// TwinCAT 3 PLC project basePLC
// ProgramVersion: 3.1.4023.0
// libraries:
//   Tc2_EtherCAT, * (Beckhoff Automation GmbH)
//   Tc2_Standard, * (Beckhoff Automation GmbH)
//   Tc2_SUPS, * (Beckhoff Automation GmbH)
//   Tc2_System, * (Beckhoff Automation GmbH)
//   Tc2_Utilities, * (Beckhoff Automation GmbH)
//   Tc3_MC2_AdvancedHoming, * (Beckhoff Automation GmbH)
//   Tc3_Module, * (Beckhoff Automation GmbH)
//   VisuDialogs, * (System)
//   Tc2_MC2,3.3.27.0,Beckhoff Automation GmbH
// project tree:
//   / GlobalTextList.TcGTLO, PlcTask.TcTTO, Visualization Manager.TcVMO (not stored)
//   GVLs/ GVL_APP.TcGVL
//   POUs/ MAIN.TcPOU
//   tc_mca_std_lib/DUTs/ RestorePosition.TcDUT, ST_AxisConfig.TcDUT, ST_AxisControl.TcDUT, MotionFunctions.TcDUT, ST_AxisInputs.TcDUT, ST_AxisPersistent.TcDUT, ST_GearAxis.TcDUT, ST_AxisStatus.TcDUT, ST_AxisStruct.TcDUT
//   tc_mca_std_lib/GVLs/ GVL.TcGVL
//   tc_mca_std_lib/POUs/ChangeConfig/ FB_ReadFloatParameter.TcPOU, FB_ReadParameterInNc_v1_00.TcPOU, FB_WriteFloatParameter.TcPOU, FB_WriteParameterInNc_v1_00.TcPOU
//   tc_mca_std_lib/POUs/ErrorHandling/ DUT_ErrorState.TcDUT, FB_ErrorSystem.TcPOU, FB_GenericError.TcPOU, FB_NC_Error.TcPOU, FB_TerminalError.TcPOU, ST_ErrorEntry.TcDUT, ST_ErrorSystem.TcDUT
//   tc_mca_std_lib/POUs/Hardware/EtherCAT_Terminals/Analog_Inputs/ EL3174_0002.TcPOU, EL3214.TcPOU, EL3255.TcPOU
//   tc_mca_std_lib/POUs/Hardware/EtherCAT_Terminals/Digital_Inputs/ EL1008.TcPOU, EL1018.TcPOU, EL1252.TcPOU, EL1808.TcPOU, EL1809.TcPOU, EL1819.TcPOU
//   tc_mca_std_lib/POUs/Hardware/EtherCAT_Terminals/Digital_Outputs/ EL2014.TcPOU, EL2252.TcPOU, EL2808.TcPOU, EL2819.TcPOU
//   tc_mca_std_lib/POUs/Hardware/EtherCAT_Terminals/Digital_Outputs/External_Types/ dutEL2521_Ctrl.TcDUT, dutEL2521_Status.TcDUT
//   tc_mca_std_lib/POUs/Hardware/EtherCAT_Terminals/Drives/ EL2522.TcPOU, EL4134.TcPOU, EL7037.TcPOU, EL7041_0052.TcPOU, EL7047.TcPOU, EL7211.TcPOU
//   tc_mca_std_lib/POUs/Hardware/EtherCAT_Terminals/Feedback_Terminals/ EL5002.TcPOU, EL5021.TcPOU, EL5042.TcPOU, EL5101.TcPOU, EL7201.TcPOU
//   tc_mca_std_lib/POUs/Hardware/EtherCAT_Terminals/System/ EK1100.TcPOU, EK1110.TcPOU, EL9410.TcPOU, EL9505.TcPOU
//   tc_mca_std_lib/POUs/Motion/ FB_Axis.TcPOU
//   tc_mca_std_lib/POUs/Motion/Homing/ FB_HomeDirect.TcPOU, FB_HomeFinish.TcPOU, FB_HomePrepare.TcPOU, FB_HomeReadNcVelocities.TcPOU, FB_HomeReadSoftLimEnable.TcPOU, FB_HomeToSwitch.TcPOU, FB_HomeVirtual.TcPOU, FB_HomeWriteNcVelocities.TcPOU, FB_HomeWriteSoftLimEnable.TcPOU, FB_Homing.TcPOU
//   tc_mca_std_lib/POUs/VISUs/ Error_Log_Visu.TcVIS, languageSupport.TcTLO, MainVisu.TcVIS, visuTextLinks.TcTLO
// (motion and I/O tree: see PLC project untitled1)
// real-time tasks:
//   TASK PlcTask: cycle T#10ms, priority 20, ADS port 350
//   TASK PlcTask1: cycle T#10ms, priority 21, ADS port 351
// variable links:

CONFIGURATION basePLC
    RESOURCE PLC ON TwinCAT3
        TASK PlcTask(INTERVAL := T#10ms, PRIORITY := 20);
        PROGRAM MAIN WITH PlcTask : MAIN;
    END_RESOURCE
END_CONFIGURATION

// ---- tc_mca_std_lib/DUTs/RestorePosition.TcDUT
{attribute 'qualified_only'}
{attribute 'strict'}
TYPE RestorePosition :
(
    DontRestore        :=0,
    RestoreWithoutHome :=1
    //RestoreWithHome    :=2
);
END_TYPE

// ---- tc_mca_std_lib/DUTs/ST_AxisConfig.TcDUT
TYPE ST_AxisConfig :
STRUCT

    ///////Axis Parameters//////
    fOverride           :   LREAL := 100;   //Controller override %
    fVelocity           :   LREAL;          //Velocity must be specified, no default used
    fAcceleration       :   LREAL;          //Not all FBs use, need to change this, 0 is NC default
    fDeceleration       :   LREAL;
    fPosition           :   LREAL;          //Used for absolute positioning
    fHomePosition       :   LREAL;          //Used to home to a value other than 0
    nHomeSeq            :   UINT;           //Homing sequence to perform
    eRestorePosition    :   RestorePosition;
    //Restore position of incremental axis after loss of power to the CPU, 0=don't restore, 1=restore but don't home, 2=restore and home

END_STRUCT
END_TYPE

// ---- tc_mca_std_lib/DUTs/ST_AxisControl.TcDUT
TYPE ST_AxisControl :
STRUCT

///////Actions from EPICS/NICOS/////////
    bExecute            :   BOOL;           //Rising edge to execute move absolute
    bReset              :   BOOL;           //Reset axis signal, must be combined with other signals
    bStop               :   BOOL;           //Stop axis movement
    bEnable             :   BOOL;           //Controller enable
    eCommand            :   MotionFunctions;

///////Axis////////
    bJogFwd             :   BOOL;           //Jog forward
    bJogBwd             :   BOOL;           //Jog backward

END_STRUCT
END_TYPE

// ---- tc_mca_std_lib/DUTs/MotionFunctions.TcDUT
{attribute 'qualified_only'}
{attribute 'strict'}
TYPE MotionFunctions :
(
    MoveAbsolute    := 0,
    MoveRelative    :=1,
    Jog             :=2,
    MoveVelocity    :=3,
    MoveModulo      :=4,
    GearIn          :=5,
    GearOut         :=6,
    MultiGearIn     :=7,
    Home            :=10
):=Jog;
END_TYPE

// ---- tc_mca_std_lib/DUTs/ST_AxisInputs.TcDUT
TYPE ST_AxisInputs :
STRUCT

///////Axis Inputs///////
    bLimitFwd   AT %I*  :   BOOL;           //Forward limit switch
    bLimitBwd   AT %I*  :   BOOL;           //Backward limit switch
    bHomeSensor AT %I*  :   BOOL;           //Reference siganl for homing
    bEncLAtch   AT %I*  :   BOOL;           //Reference index signal from inc. enconder

END_STRUCT
END_TYPE

// ---- tc_mca_std_lib/DUTs/ST_AxisPersistent.TcDUT
TYPE ST_AxisPersistent :
STRUCT

    PERSISTENT iPositionAtShutdown : LREAL;
    bMovingAtShutdown   : BOOL;

END_STRUCT
END_TYPE

// ---- tc_mca_std_lib/DUTs/ST_GearAxis.TcDUT
TYPE ST_GearAxis :
STRUCT
    index   :   UINT:=1;    //index of master axis
    ratio   :   LREAL;      //gearing ratio
END_STRUCT
END_TYPE

// ---- tc_mca_std_lib/DUTs/ST_AxisStatus.TcDUT
TYPE ST_AxisStatus :
STRUCT

///////Outputs/Status/////////
    bEnabled            :   BOOL;           //Axis drive enabled
    bWarning            :   BOOL;           //Warning violation (need to be deinfed all the warning stages)
    bBusy               :   BOOL;           //Axis busy
    bDone               :   BOOL;           //Last function block executed successfully
    bHomed              :   BOOL;           //Axis homed
    bFwEnabled          :   BOOL;           //Positive movement of axis is enabled/disabled
    bBwEnabled          :   BOOL;           //Negative movement of axis is enabled/disabled
    fActPosition        :   LREAL;          //Actual position value
    fActVelocity        :   LREAL;          //Actual velocity
    bError              :   BOOL;           //Motion function block has produced error (NC drive not necessarily in error state)
    nErrorID            :   UDINT;          //Motion function block errorID
    bGeared             :   BOOL;           //Axis is an active slave

END_STRUCT
END_TYPE

// ---- tc_mca_std_lib/DUTs/ST_AxisStruct.TcDUT
TYPE ST_AxisStruct :
STRUCT

///////Actions from EPICS/NICOS/////////
///////Axis////////
    control     : ST_AxisControl;

///////Outputs/Status/////////
    status      : ST_AxisStatus;

///////Axis Parameters//////
    config      : ST_AxisConfig;

///////Axis Inputs///////
    inputs      : ST_AxisInputs;

//////Geraing Parameters//////
    //masterAxis        :   UINT:=1;        //Axes[ ] index for master
    //fGearRatioNum     :   LREAL;          //GearIn ratio numerator
    //iGearRatioDen     :   UINT;           //GearIn ratio denominator
///////Axis Ref/////
    Axis                :   AXIS_REF;       //Link NC axis to this

    masterAxis          :   ST_GearAxis;    //Single master axis
    //slaveAxis         :   ARRAY [1..GVL.axisNum]OF ST_GearAxis :=(index:=0, ratio:=0) ;   //Linking single slave axes
    slaveAxisRatio      :   ARRAY [1..GVL_APP.axisNum] OF LREAL;


//////Extra things of original ISIS Structure/////

    //  bSoftLimPosEn       :   BOOL;           //Enable/disable positive direction software limit
    //  bSoftLimNegEn       :   BOOL;           //Enable/disable negative direction software limit
    //bPosLagEn         :   BOOL;           //Enable/disable position lag

    //Gearing parameters

    //masterAxes            :   ARRAY[1..4] OF ST_MasterAxis;   //ST to hold index and ratio for masters    - GearInMultiMaster
    //fDeceleration     :   LREAL;          //Not all FBs use, need to change this, 0 is NC default
    //  Status              : ST_AxisStatus;
END_STRUCT
END_TYPE

// ---- tc_mca_std_lib/POUs/ErrorHandling/DUT_ErrorState.TcDUT
{attribute 'qualified_only'}
{attribute 'strict'}
TYPE DUT_ErrorState :
(
    None,
    Active,
    Inactive,
    Acknowledged
);
END_TYPE

// ---- tc_mca_std_lib/POUs/ErrorHandling/ST_ErrorEntry.TcDUT
TYPE ST_ErrorEntry :
STRUCT
    ErrorNum    : ULINT := 0;               //ID of the Error entry
    ErrorState  : DUT_ErrorState;           //State of the error

    //Error related
    iTerminalID     : INT;                  //ID of the terminal
    sDateTimeOn     : STRING(24);           //Date and time when the error occured
    sDateTimeOff    : STRING(24);           //Date and time when the error disapeared
    sErrorMessage   : STRING (128);         //Description of the event

    ErrorPriority   : INT;                  //Priority of the error
END_STRUCT
END_TYPE

// ---- tc_mca_std_lib/POUs/ErrorHandling/ST_ErrorSystem.TcDUT
TYPE ST_ErrorSystem :
STRUCT
    //Array of error data. Size = cSizeOfErrorData in the GVL
    aErrorData      : ARRAY [0..cSizeOfErrorData - 1] OF ST_ErrorEntry;     //Error Entry List
    nNextErrorNum   : ULINT := 1;                   //ErrorID for the next error entry
    nNoError        : UINT;                         //Number of errors in the list
    nNoActive       : UINT;                         //Number of Active errors
    nNoInactive     : UINT;                         //Number on Inactive errors
    nNoFree         : UINT;                         //Number of free entries in the list
    nNoOverflow     : INT := 0;                     //Number of overflows. How many error entries have been lost due to the size of the array
END_STRUCT
END_TYPE

// ---- tc_mca_std_lib/POUs/Hardware/EtherCAT_Terminals/Digital_Outputs/External_Types/dutEL2521_Ctrl.TcDUT
TYPE dutEL2521_Ctrl :
STRUCT
    ///The control word (CW) is located in the output process image, and is transmitted from the controller to the terminal.
    ///CW.0 FREQ_SEL 0bin / 1bin  Rapid change of the base frequency (only if the ramp function is inactive):
    ///0bin = Base frequency 1 (object 8001:02)
    ///1bin = Base frequency 2 (object 8001:03)
    FREQ_SEL: BOOL;
    ///CW.1 RAMP_DIS 1bin Operation of the ramp function is cancelled, in spite of object 8000:06 being active; if travel distance control is active, it is interrupted by this bit
    RAMP_DIS: BOOL;
    ///CW.2 GO_COUNTER 1bin  If travel distance control is active (object 8000:0A), then a pre-set counter value is approached when the bit is set
    GO_COUNTER: BOOL;
    ///CW.5 CNT_CLR 1bin The contents of the counter is cleared or set (object 8000:0B) by this bit.
    ///Any overflow or underflow bits that might be set are also cleared by this bit.
    ///The process can be edge triggered or level triggered (object 8000:05).
    CNT_CLR: BOOL;
END_STRUCT
END_TYPE

// ---- tc_mca_std_lib/POUs/Hardware/EtherCAT_Terminals/Digital_Outputs/External_Types/dutEL2521_Status.TcDUT
TYPE dutEL2521_Status :
STRUCT
    ///The status word (SW) is located in the input process image, and is transmitted from the terminal to the controller.
    ///SW.0 SEL_ACK/END_COUNTER 1bin  Confirms the change of base frequency. At activated travel distance control: target counter value reached
    SEL_ACK: BOOL;
    ///SW.1 RAMP_ACTIVE 1bin Ramp is currently being followed
    RAMP_ACTIVE: BOOL;
    ///SW.2 UNDERFLOW 1bin This bit is set if the 16-bit counter underflows (0 -> 65535). It is reset when the counter drops below two thirds of its measuring range (43690 -> 43689) or immediately an overflow occurs.
    UNDERFLOW: BOOL;
    ///SW.3 OVERFLOW 1bin This bit is set if the 16-bit counter overflows (65535 -> 0). It is reset when the counter exceeds one third of its measuring range (21845 -> 21846) or immediately an underflow occurs
    OVERFLOW: BOOL;
    ///SW.4 INPUT_T 1bin Status of INPUT_T
    INPUT_T: BOOL;
    ///SW.5 INPUT_Z 1bin Status of INPUT_Z
    INPUT_Z: BOOL;
    ///SW.6 ERROR 1bin General error bit, included with overflow/underflow
    ERROR: BOOL;
END_STRUCT
END_TYPE

// ---- GVLs/GVL_APP.TcGVL
{attribute 'qualified_only'}
VAR_GLOBAL

END_VAR

VAR_GLOBAL CONSTANT
    axisNum :   UINT:=2;
    //axisCoupleMax :   UINT:=4;
END_VAR

// ---- tc_mca_std_lib/GVLs/GVL.TcGVL
VAR_GLOBAL
    stErrorSystemCom    : ST_ErrorSystem;
    axes            :   ARRAY [1..GVL_APP.axisNum] OF ST_AxisStruct;    //Global array of axisControl structure for holding axis parameters and controls
    iAxis           :   UINT;                                           //Index for running axis

END_VAR

VAR_GLOBAL CONSTANT
    cSizeOfErrorData : UINT := 256;
END_VAR

VAR_GLOBAL PERSISTENT
    axesPersistent  : ARRAY [1..gvl_app.axisNum] OF ST_AxisPersistent;
END_VAR

// ---- POUs/MAIN.TcPOU
PROGRAM MAIN
VAR
    sVersion: STRING:='1.0.0';
    i : UINT; //index variable for AXES()
    aFbAxes: ARRAY [1..gvl_app.axisNum] OF FB_Axis;
    hmiAxisSelection    :   INT:=1;     //Not possible to use local hmi variables for array indexes

(******Outputs: Power for Limit switches and Home Sensors (every 4th output)********)

    bOutput1 AT %Q*: BOOL:= TRUE;
    //bOutput2 AT %Q*: BOOL:= TRUE;
    //bOutput3 AT %Q*: BOOL:= TRUE;
    //bOutput4 AT %Q*: BOOL:= TRUE;
    //bOutput5 AT %Q*: BOOL:= TRUE;
    //bOutput6 AT %Q*: BOOL:= TRUE;
    //bOutput7 AT %Q*: BOOL:= TRUE;
    //bOutput8 AT %Q*: BOOL:= TRUE;
    //bOutput9 AT %Q*: BOOL:= TRUE;
    //bOutput13 AT %Q*: BOOL:= TRUE;
    //bOutput17 AT %Q*: BOOL:= TRUE;
    //bOutput21 AT %Q*: BOOL:= TRUE;
    //bOutput24 AT %Q*: BOOL:= TRUE;
    //bOutput28 AT %Q*: BOOL:= TRUE;

(******Error Handling********)
    fbErrorSystem: FB_ErrorSystem;
    aFbAxesError: ARRAY [1..gvl_app.axisNum] OF FB_NC_Error;

    //fbEL1018  : EL1018;
    //fbEL2808  : EL2808;
    //fbEL5101  : EL5101;
    //fbEL9505  : EL9505;
    //fbEL1252  : EL1252;
    //fbEL9410  : EL9410;
    //fbEL7037  : EL7037;
    //fbEK1110  : EK1110;

(******Startup, Shutdown and UPS********)
    fbUPS                  : FB_S_UPS_CX51x0;
    eUpsMode               : E_S_UPS_Mode   := eSUPS_WrPersistData_Shutdown;
    eStartUp: (ColdStart, ReadAxisFeedbackType, CheckReadDone, ExecuteRestore, CheckRestore, FinishRestore);
    bPositionRestoreDone   : BOOL := FALSE;
    bRestoreExecute        : BOOL := FALSE;
    bExecuteReadEncRefSys  : BOOL := FALSE;
    iRetry                 : INT;
    fbReadEncRefSys        : ARRAY [1..gvl_app.axisNum] OF MC_ReadParameter;
    fbRestorePosition      : ARRAY [1..GVL_app.axisNum] OF MC_SetPosition;

END_VAR

VAR PERSISTENT
    bRestoreOnStartup : BOOL;
END_VAR

fbUPS(eUpsMode := eUpsMode); (* call UPS-FB instance in first lines of the fastest PLC Task *)

IF eGlobalSUpsState = eSUPS_PowerFailure THEN
    (* first cycle of powerfailure *)
    (* execute code that should only be done once with each powerfailure, i.e. increase powerfailure counter *)
    bRestoreOnStartup:=TRUE;
    STORE_PERSISTENT();
    RETURN;
ELSIF eGlobalSUpsState > eSUPS_PowerFailure THEN
    (* next cycles of powerfailure *)
    (* skip regular code execution for the remaining cycles of the powerfailure/writing of persistent data/quick shutdown  ... *)
    RETURN;
END_IF

RESTORE_POSITIONS();
PROG();
AXES();
ERROR();

ACTION AXES:
FOR GVL.iAxis:=1 TO gvl_app.axisNum DO
    aFbAxes[GVL.iAxis](stAxisStruct:=gvl.axes[GVL.iAxis]);
END_FOR
END_ACTION

ACTION ERROR:
//
(****FB containting the log of the errors****)
//
fbErrorSystem(
    En:= TRUE,
    bReset:= ,
    nErrorNum:= ,
    bACK:= ,
    bValidSelection:= ,
    nTableRowIndex:= ,
    EnO=> ,
    nSelectedError=> ,
    pErrorSystem=> );


FOR GVL.iAxis:=1 TO gvl_app.axisNum DO
    aFbAxesError[gvl.iAxis](EN:=TRUE,
    nNC_ErrorID:= gvl.axes[gvl.iAxis].status.nErrorID,
    nNC_AxisID:=gvl.axes[gvl.iAxis].Axis.NcToPlc.AxisId,
    ErrorSystem:= fbErrorSystem.pErrorSystem);
END_FOR



(*call all the necessary instance (input assistance F2 or right click) according to the terminals that you have in your hardware and
 add "TRUE" in the input En, the corresponding number of termianl to the iTerminal_ID and
the variable "fbErrorSystem.pErrorSystem" to the input ErrorSystem in each FB E. g. :
fbEL1808(
    En:= TRUE,
    iTerminal_ID:= 01,
    ErrorSystem:= fbErorSystem.pErrorSystem,
    EnO=> ,
    bError=> );
 *)
END_ACTION

ACTION PROG:
//
(* Program any sequence, safety or feature (if necessary) application specific in thsi section*)

//
END_ACTION

ACTION RESTORE_POSITIONS:
///#########################################################
// This ACT will restore the position of an incremental axis on startup with the act position it read before losing power.
// It checks the type of axis, 0=incremental, and that the axis was stationary at shut down.
// Because 0 equates to incremental we also need to check that the data is valid, otherwise by default it would restore all axes.
// By default an axis will not restore the position unless it is set to opt-in, i.e. gvl.axes[i].config.eRestorePosition is non-zero.
// This needs to be initialised somewhere in TwinCAT code otherwise it will not be available at start up.
// A restore will only be performed on a loss of power, this code shouldn't make any changes on a reset cold, a rest origin or a download.
// There is a enum to allow for different types of restore modes, currently only one is implemented.
// 0 'DontRestore'
// 1 'RestoreWithoutHome' -restores the position using a set position fb and does not set the home bit in the axis struct.
// Note from Beckhoff: "A maximum of 1 MB persistent data can be reliably saved over the entire service life."
///#########################################################

IF bRestoreOnStartup THEN
    bRestoreOnStartup:=FALSE;
    bRestoreExecute:=TRUE;
END_IF

// Upon startup bPositionRestoreDone will be set to FALSE, after successfully completing the following code it will be set TRUE
// and should stay TRUE for the rest of the time the PLC is operational, thus this routine should only be completed once.
IF bRestoreExecute AND NOT bPositionRestoreDone THEN

    // Cycle through function blocks that read the encoder reference system i.e. whether axis is incremental or absolute
    // Result stored in Value, 0=Inc 1=Abs, execute set during the case statement
    FOR i:=1 TO gvl_app.axisNum DO
        fbReadEncRefSys[i](
          Axis:= gvl.axes[i].Axis,
          Enable:= bExecuteReadEncRefSys,
          ParameterNumber:= MC_AxisParameter.AxisEncoderReferenceSystem,
          Value=>,
          ReadMode:= E_READMODE.READMODE_ONCE);
    END_FOR

    // Cycle through set position function blocks for each axis
    FOR i:=1 TO gvl_app.axisNum DO
        fbRestorePosition[i](
         Axis:= gvl.axes[i].Axis,
         Execute:= ,
         Position:= axesPersistent[i].iPositionAtShutdown);
    END_FOR

    CASE eStartUp OF
        ColdStart:
        // First cycle of the PLC, do nothing just give one cycle for variables to initialise
            IF NOT bPositionRestoreDone THEN
                eStartUp:=eStartUp+1;
                iRetry:=0;
            END_IF

        ReadAxisFeedbackType:
        // Exectute the function blocks to read the encoder reference system (0=inc OR 1=ABS)
            bExecuteReadEncRefSys:=TRUE;
            eStartUp:=eStartUp+1;

        CheckReadDone:
        // Check the encoder reference system has been read for all axis -> if busy then continue with PLC cycle and check again next time.
        // If fbReadEncRefSys not started then go back a step.
        // If any axes result in an error the code will get stuck here, this happens if gvl_app.axisNum is not set correctly
            FOR i:=1 TO gvl_app.axisNum DO
                IF fbReadEncRefSys[i].Valid = FALSE THEN
                    IF fbReadEncRefSys[i].Busy = TRUE THEN
                        // Exit MAIN.STARTUP Action and wait till next cycle, needs to cycle through whole program in order for data to update
                        RETURN;
                    ELSE
                        // Sometimes the code gets here and the fbReadEncRefSys[i] misses the rising edge. If  the code gets here it means
                        // .valid=FALSE and .busy=FALSE which indicateds the FB probably hasn't started and thus needs to see a rising edge.
                        // Set execute to low, Exit MAIN.STARTUP and go back a step in the CASE statement.
                        bExecuteReadEncRefSys:=FALSE;
                        eStartUp:=eStartUp-1;
                        iRetry:=iRetry+1; // counter used for troubleshooting to see how many cycles it takes before fbReadEncRefSys function blocks are read correctly
                        RETURN;
                    END_IF
                END_IF
            END_FOR
            // If the code gets here all axes either have .valid=TRUE for all axes
            eStartUp:=eStartUp+1;

        ExecuteRestore:
        // Execute position restore by setting fbRestorePosition.execute = TRUE
            FOR i:=1 TO gvl_app.axisNum DO
                IF fbReadEncRefSys[i].Valid = TRUE AND fbReadEncRefSys[i].Value = 0 AND NOT(axesPersistent[i].bMovingAtShutdown) THEN
                    IF GVL.axes[i].config.eRestorePosition = RestorePosition.RestoreWithoutHome THEN
                        fbRestorePosition[i].Execute:=TRUE;
                    END_IF
                END_IF
            END_FOR
            eStartUp:=eStartUp+1;

        CheckRestore:
        // Check the set position fbs are finished
        // Nothing actually happens if the restore is not done, the code just returns from here each cycle and the
        // bPositionRestoreDone will never get set to TRUE and will take up cycle time
            FOR i:=1 TO gvl_app.axisNum DO
                IF fbReadEncRefSys[i].Valid = TRUE AND fbReadEncRefSys[i].Value = 0 AND NOT(axesPersistent[i].bMovingAtShutdown) THEN
                    IF GVL.axes[i].config.eRestorePosition = RestorePosition.RestoreWithoutHome THEN
                        IF NOT fbRestorePosition[i].Done THEN
                            RETURN;
                        END_IF
                    END_IF
                END_IF
            END_FOR
            eStartUp:=eStartUp+1;

        FinishRestore:
        // Remove execute = TRUE for fbRestorePosition
            FOR i:=1 TO gvl_app.axisNum DO
                fbRestorePosition[i].Execute:=FALSE;
            END_FOR
            bPositionRestoreDone:=TRUE;
            bRestoreExecute:=FALSE;
    END_CASE
END_IF
END_ACTION

ACTION STORE_PERSISTENT:
FOR i:=1 TO gvl_app.axisNum DO
    axesPersistent[i].iPositionAtShutdown:=gvl.axes[i].Axis.NcToPlc.ActPos;
    IF gvl.axes[i].Axis.NcToPlc.ActVelo <> 0 THEN
        axesPersistent[i].bMovingAtShutdown:=TRUE;
    ELSE
        axesPersistent[i].bMovingAtShutdown:=FALSE;
    END_IF
    axesPersistent[i].bMovingAtShutdown:=axesPersistent[i].bMovingAtShutdown OR gvl.axes[i].Axis.Status.Moving;
END_FOR
END_ACTION

END_PROGRAM

// ---- tc_mca_std_lib/POUs/Motion/FB_Axis.TcPOU
///#########################################################
///Function block to run a virtual drive with Nc
/// Library:
/// Tc2_MC2.lib
///
/// Global Variables:
///
/// Data types:
///
/// External functions:
///
///###########################################################
FUNCTION_BLOCK FB_Axis
VAR
    sVersion: STRING:='1.0.4';
    masterAxis          :   ST_GearAxis :=(index:=1, ratio:=0) ;

    i: UINT;
END_VAR
VAR_INPUT

END_VAR
VAR_OUTPUT

END_VAR

VAR_IN_OUT
    stAxisStruct: ST_AxisStruct;
END_VAR
VAR
    fbReset: MC_Reset;
    fbPower: MC_Power;
    fbStop: MC_Stop;
    fbHalt: MC_Halt;
    fbJog: MC_Jog;
    fbMoveAbsolute: MC_MoveAbsolute;
    fbMoveVelocity: MC_MoveVelocity;
    fbMoveRelative: MC_MoveRelative;
    fbMoveModulo: MC_MoveModulo;
    fbGearIn: MC_GearIn;
    fbGearOut: MC_GearOut;
    fbHome: FB_Homing;
    fbExecuteRiseEdge: R_TRIG;
    fbStopRiseEdge: R_TRIG;
    fbResetRiseEdge: R_TRIG;
END_VAR

stAxisStruct.Axis.ReadStatus();

////Call of all MC Instances//////

fbPower(Axis:=stAxisStruct.Axis);
fbPower.Enable:= FALSE;
fbReset(Axis:=stAxisStruct.Axis);
fbReset.Execute:= FALSE;
fbStop(Axis:=stAxisStruct.Axis);
fbStop.Execute:=FALSE;
fbHalt(Axis:=stAxisStruct.Axis);
fbHalt.Execute:=FALSE;
fbJog(Axis:=stAxisStruct.Axis);
fbHome(Axis:=stAxisStruct.Axis);
fbHome.bExecute:=FALSE;
fbMoveAbsolute(Axis:=stAxisStruct.Axis);
fbMoveAbsolute.Execute:=FALSE;
fbMoveRelative(Axis:=stAxisStruct.Axis);
fbMoveRelative.Execute:=FALSE;
fbMoveVelocity(Axis:=stAxisStruct.Axis);
fbMoveVelocity.Execute:=FALSE;
fbMoveModulo(Axis:=stAxisStruct.Axis);
fbMoveModulo.Execute:=FALSE;
fbGearin(Slave:= stAxisStruct.Axis, Master:= GVL.axes[masterAxis.index].Axis);
fbGearIn.Execute:=FALSE;
fbGearOut(Slave:=stAxisStruct.Axis);
fbGearOut.Execute:=FALSE;

stAxisStruct.status.bFwEnabled:= stAxisStruct.inputs.bLimitFwd;
stAxisStruct.status.bBwEnabled:= stAxisStruct.inputs.bLimitBwd;

FOR i:= 1 TO GVL_APP.axisNum DO
    IF (stAxisStruct.slaveAxisRatio[i]<>0) THEN
        stAxisStruct.status.bFwEnabled:=stAxisStruct.status.bFwEnabled AND SEL(stAxisStruct.slaveAxisRatio[i]>0, GVL.axes[i].status.bBwEnabled, GVL.axes[i].status.bFwEnabled);
        stAxisStruct.status.bBwEnabled:=stAxisStruct.status.bBwEnabled AND SEL(stAxisStruct.slaveAxisRatio[i]>0, GVL.axes[i].status.bFwEnabled, GVL.axes[i].status.bBwEnabled);
    END_IF
END_FOR

(*Power*)
    fbPower.Enable:=stAxisStruct.control.bEnable;
    fbPower.Enable_Positive:= stAxisStruct.status.bFwEnabled;
    fbPower.Enable_Negative:= stAxisStruct.status.bBwEnabled;
    fbPower.Override:= stAxisStruct.config.fOverride;
    stAxisStruct.status.bEnabled:=fbPower.Status;

(*Stop*)
    fbStop.Execute:= stAxisStruct.control.bStop;
    fbStop.Deceleration:= stAxisStruct.config.fDeceleration;

IF stAxisStruct.control.bStop AND stAxisStruct.Axis.Status.Stopping THEN
    stAxisStruct.control.bStop:=FALSE;
END_IF

(*Reset*)
    fbReset.Execute:=stAxisStruct.control.bReset AND stAxisStruct.status.bError;

IF stAxisStruct.control.bReset AND NOT (stAxisStruct.status.bError OR stAxisStruct.status.bWarning) THEN
    stAxisStruct.control.bReset:=FALSE;
END_IF

CASE stAxisStruct.control.eCommand OF
    MotionFunctions.MoveAbsolute:
        fbMoveAbsolute.Execute:=stAxisStruct.control.bExecute;
        fbMoveAbsolute.Position:=stAxisStruct.config.fPosition;
        fbMoveAbsolute.Velocity:=ABS(stAxisStruct.config.fVelocity);
        fbMoveAbsolute.Acceleration:=stAxisStruct.config.fAcceleration;
        fbMoveAbsolute.Deceleration:=stAxisStruct.config.fDeceleration;

    MotionFunctions.MoveRelative:
        fbMoveRelative.Execute:=stAxisStruct.control.bExecute;
        fbMoveRelative.Distance:=stAxisStruct.config.fPosition;
        fbMoveRelative.Velocity:=ABS(stAxisStruct.config.fVelocity);
        fbMoveRelative.Acceleration:=stAxisStruct.config.fAcceleration;
        fbMoveRelative.Deceleration:=stAxisStruct.config.fDeceleration;

    MotionFunctions.Jog:
        fbJog.JogForward:=stAxisStruct.control.bJogFwd AND NOT (stAxisStruct.control.bExecute OR stAxisStruct.status.bError);
        fbJog.JogBackwards:=stAxisStruct.control.bJogBwd AND NOT (stAxisStruct.control.bExecute OR stAxisStruct.status.bError);
        fbJog.Mode:=0;
        fbJog.Velocity:=stAxisStruct.config.fVelocity;
        fbJog.Acceleration:=stAxisStruct.config.fAcceleration;
        fbJog.Deceleration:=stAxisStruct.config.fDeceleration;

    MotionFunctions.MoveVelocity:
        fbMoveVelocity.Execute:=stAxisStruct.control.bExecute;
        fbMoveVelocity.Velocity:=ABS(stAxisStruct.config.fVelocity);
        fbMoveVelocity.Acceleration:=stAxisStruct.config.fAcceleration;
        fbMoveVelocity.Deceleration:=stAxisStruct.config.fDeceleration;
        fbMoveVelocity.Direction:=SEL(stAxisStruct.config.fVelocity<0, MC_Positive_Direction, MC_Negative_Direction);

    MotionFunctions.Movemodulo:
        fbMoveModulo.Execute:=stAxisStruct.control.bExecute;
        fbMoveModulo.Position:=stAxisStruct.config.fPosition;
        fbMoveModulo.Velocity:=ABS(stAxisStruct.config.fVelocity);
        fbMoveModulo.Acceleration:=stAxisStruct.config.fAcceleration;
        fbMoveModulo.Deceleration:=stAxisStruct.config.fDeceleration;


    MotionFunctions.GearIn:
        fbGearIn.Execute:=          stAxisStruct.control.bExecute;
        fbGearIn.RatioNumerator:=   masterAxis.Ratio;
        fbGearIn.RatioDenominator:=1;       //kept static as numerator is LREAL and consistent with multigearing

        IF NOT fbGearIn.InGear THEN
            masterAxis.Index:=  stAxisStruct.masterAxis.index;
            masterAxis.Ratio:= stAxisStruct.masterAxis.ratio;
        END_IF

        IF fbGearIn.InGear AND (GVL.axes[masterAxis.Index].slaveAxisRatio[GVL.iAxis]=0) THEN    //only update index and ratios on new gearIns, change of ratio requires gearOut
            GVL.axes[masterAxis.index].slaveAxisRatio[GVL.iAxis]:=masterAxis.ratio;
        END_IF

    MotionFunctions.GearOut:
        fbGearOut.Execute:=         stAxisStruct.control.bExecute;

        IF fbGearOut.Done THEN
            GVL.axes[masterAxis.index].slaveAxisRatio[GVL.iAxis]:=0; //Clear slave ratio from master axis slave array
        END_IF

    MotionFunctions.MultiGearIn:

    MotionFunctions.Home:
        fbHome.bExecute:= stAxisStruct.control.bExecute;
        fbHome.bReset:= stAxisStruct.control.bReset;
        fbHome.bStop:= stAxisStruct.control.bStop;
        fbHome.nHomeProc:= stAxisStruct.config.nHomeSeq;
        fbHome.fHomePosition:= stAxisStruct.config.fHomePosition;
        fbHome.bLimitBwd:= stAxisStruct.inputs.bLimitBwd;
        fbHome.bLimitFwd:= stAxisStruct.inputs.bLimitFwd;
        fbHome.bEncLatch:= stAxisStruct.inputs.bEncLatch;
        fbHome.bHomeSensor:= stAxisStruct.inputs.bHomeSensor;
        fbHome.fHomePosition:= 0;
        stAxisStruct.status.bHomed:=fbHome.bHomed;

END_CASE

(*Busy*)
stAxisStruct.status.bBusy:=stAxisStruct.Axis.Status.HasJob;

(*Done*)
IF fbMoveAbsolute.Done OR fbMoveModulo.Done OR fbMoveRelative.Done THEN
        stAxisStruct.status.bDone:=TRUE;
ELSIF stAxisStruct.Axis.Status.HasJob THEN
        stAxisStruct.status.bDone:=FALSE;
END_IF

(*Error from functions and Nc*)
IF stAxisStruct.status.bError and not stAxisStruct.control.bReset THEN
    stAxisStruct.status.bError:=stAxisStruct.status.bError;
    stAxisStruct.status.nErrorID:=stAxisStruct.status.nErrorID;
ELSIF fbPower.Error THEN
    stAxisStruct.status.bError:=TRUE;
    stAxisStruct.status.nErrorId:=fbPower.ErrorID;
ELSIF fbHalt.Error THEN
    stAxisStruct.status.bError:=TRUE;
    stAxisStruct.status.nErrorId:=fbHalt.ErrorID;
ELSIF fbJog.Error THEN
    stAxisStruct.status.bError:=TRUE;
    stAxisStruct.status.nErrorId:=fbJog.ErrorID;
ELSIF fbMoveVelocity.Error THEN
    stAxisStruct.status.bError:=TRUE;
    stAxisStruct.status.nErrorId:=fbMoveVelocity.ErrorID;
ELSIF fbMoveRelative.Error THEN
    stAxisStruct.status.bError:=TRUE;
    stAxisStruct.status.nErrorId:=fbMoveRelative.ErrorID;
ELSIF fbMoveAbsolute.Error THEN
    stAxisStruct.status.bError:=TRUE;
    stAxisStruct.status.nErrorId:=fbMoveAbsolute.ErrorID;
ELSIF fbMoveModulo.Error THEN
    stAxisStruct.status.bError:=TRUE;
    stAxisStruct.status.nErrorId:=fbMoveModulo.ErrorID;
ELSIF fbHome.bError THEN
    stAxisStruct.status.bError:=TRUE;
    stAxisStruct.status.nErrorId:=fbHome.nErrorID;
ELSIF fbGearIn.Error THEN
    stAxisStruct.status.bError:=TRUE;
    stAxisStruct.status.nErrorId:=fbGearIn.ErrorID;
ELSIF fbGearIn.Error THEN
    stAxisStruct.status.bError:=TRUE;
    stAxisStruct.status.nErrorId:=fbGearIn.ErrorID;
ELSIF fbGearOut.Error and stAxisStruct.Axis.Status.Coupled THEN
    stAxisStruct.status.bError:=TRUE;
    stAxisStruct.status.nErrorId:=fbGearOut.ErrorID;
ELSIF stAxisStruct.Axis.Status.Error  THEN
    stAxisStruct.status.bError:=stAxisStruct.Axis.Status.Error;
    stAxisStruct.status.nErrorId:=stAxisStruct.Axis.Status.ErrorID;
ELSE
    stAxisStruct.status.bError:=FALSE;
    stAxisStruct.status.nErrorId:=0;
END_IF;

(*Warnings from functions and Nc*)
IF stAxisStruct.status.bWarning AND NOT stAxisStruct.control.bReset THEN
    stAxisStruct.status.bWarning:=stAxisStruct.status.bWarning;
    //stAxisStruct.status.nWarningID:=stAxisStruct.status.nWarningID;
ELSIF fbHome.bWarning THEN
    stAxisStruct.status.bWarning:=stAxisStruct.status.bError;
    //stAxisStruct.status.nWarningID:=stAxisStruct.status.nWarningID;
ELSE
    stAxisStruct.status.bWarning:=FALSE;
    //stAxisStruct.status.nWarningId:=0;
END_IF;

stAxisStruct.status.bGeared:= stAxisStruct.Axis.Status.Coupled;

(*Actual Velocity*)
stAxisStruct.status.fActVelocity:=stAxisStruct.Axis.NcToPlc.ActVelo;

(*Actual Position*)
IF stAxisStruct.Axis.Status.OpMode.Modulo THEN
    stAxisStruct.status.fActPosition:=stAxisStruct.Axis.NcToPlc.ModuloActPos;
ELSE
    stAxisStruct.status.fActPosition:=stAxisStruct.Axis.NcToPlc.ActPos;
END_IF

(*Reset bExecute*)
stAxisStruct.control.bExecute:=FALSE;

END_FUNCTION_BLOCK

// ---- tc_mca_std_lib/POUs/Motion/Homing/FB_Homing.TcPOU
FUNCTION_BLOCK FB_Homing
VAR_INPUT
    bExecute: BOOL;
    bReset: BOOL;
    bStop: BOOL;
    nHomeProc: UINT;
    bLimitBwd: BOOL;
    bLimitFwd: BOOL;
    bEncLatch: BOOL;
    bHomeSensor: BOOL;
    fHomePosition: LREAL;
END_VAR
VAR_IN_OUT
    Axis: AXIS_REF;
END_VAR
VAR_OUTPUT
    bHomed:BOOL;
    bError: BOOL;
    bWarning: BOOL;
    nErrorId: UDINT;
END_VAR
VAR
    bHomingInProgress: BOOL;
    bReadNCVelocities: BOOL;
    nHomeProcLocal: UINT := 0;
    nHomingState: INT := 0;
    fbExecuteRiseEdge: R_TRIG;
    fbHomingParameter: MC_HomingParameter;
    fbRef_Signal_Ref1: MC_Ref_Signal_Ref;
    fbRef_Signal_Ref2: MC_Ref_Signal_Ref;
    fbRef_Signal_Ref3: MC_Ref_Signal_Ref;
    fbRef_Signal_Ref4: MC_Ref_Signal_Ref;
    StOptions2: ST_Home_Options2;
    StOptions4: ST_Home_Options4;
    tLimit: TIME :=  T#0H10M;
    fbStepLimitSwitch: MC_StepLimitSwitch;
    fbStepLimitSwitchDetection: MC_StepLimitSwitchDetection;
    fbStepAbsoluteSwitch: MC_StepAbsoluteSwitch;
    fbStepReferencePulse: MC_StepReferencePulse;
    fbHomeDirect: MC_HomeDirect;
    fbAbortHoming: MC_AbortHoming;
    fbFinishHoming: MC_FinishHoming;
    fbHomeReadNCVelocities: FB_HomeReadNCVelocities;

    trigger: TRIGGER_REF;
    touchProbe: MC_TouchProbe;
END_VAR

IF bReset THEN
    bError:=FALSE;
    bWarning:=FALSE;
    bReadNCVelocities:=FALSE;
    bHomingInProgress:=FALSE;
    fbAbortHoming.Execute:=FALSE;
    nErrorId:=0;
    nHomingState:=0;
END_IF

IF bStop THEN
    //fbAbortHoming.Execute:=TRUE;
    bReadNCVelocities:=FALSE;
    bHomingInProgress:=FALSE;
    nHomingState:=0;
END_IF

fbExecuteRiseEdge(CLK:=bExecute);
IF fbExecuteRiseEdge.Q THEN
    bHomingInProgress:=TRUE;
    bReadNCVelocities:=TRUE;
    fbAbortHoming.Execute:=FALSE;
    nHomeProcLocal:=nHomeProc;
    CASE nHomeProcLocal OF
      //0X: LIMIT Switch
      01: //Home to bBwdLimit (reverse off limit)
      02: //Home to bFwdLimit (reverse off limit)
      03: //Home to bBwdLimit (two speeds)
      04: //Home to bFwdLimit (two speeds)
      //1X: Home Sensor
      11: //Home to bHome in Bwd direction (single speed - will reverse back if limit hit)
      12: //Home to bHome in Fwd direction (single speed - will reverse back if limit hit)
      13: //Home to bHome via bBwdLimit (two speeds)
      14: //Home to bHome via bFwdLimit (two speeds)
      //2X: Enc Pulse
      21: //Home to EncRefPulse in Bwd direction (single speed - will reverse back if limit hit)
      22: //Home to EncRefPulse in Fwd direction (single speed - will reverse back if limit hit)
      23: //Home to EncRefPulse via bBwdLimit (two speeds)
      24: //Home to EncRefPulse via bFwdLimit (two speeds)
      //9X: Software
      90: //Home direct to value
    ELSE
      bError:=TRUE;
      bHomingInProgress := FALSE;
      nErrorId:=16#4FFF;
  END_CASE
END_IF

IF bHomingInProgress AND fbHomeReadNCVelocities.bDone AND NOT bError THEN
CASE nHomeProcLocal OF
   1,2: //Home to bLimitBwd(1) or bLimitFwd(2)
        CASE nHomingState OF
          0:
            fbStepLimitSwitch.Execute:=FALSE;
            fbStepLimitSwitch.LimitSwitchMode:=mcFallingEdge;
            fbStepLimitSwitch.Velocity:=fbHomeReadNCVelocities.fVelocityFromCam;
            fbStepLimitSwitch.Setposition:=fHomePosition;
            CASE nHomeProcLocal OF
                1: fbStepLimitSwitch.Direction:=mcNegativeDirection;
                2: fbStepLimitSwitch.Direction:=mcPositiveDirection;
            END_CASE
            nHomingState:=nHomingState+1;
          1:
            fbStepLimitSwitch.Execute:=TRUE;
            nHomingState:=nHomingState+1;
          2:
            IF fbStepLimitSwitch.Busy THEN
                nHomingState:=nHomingState+1;
            END_IF
          3:
            IF fbStepLimitSwitch.Done THEN
                fbFinishHoming.Execute:=TRUE;
                nHomingState:=nHomingState+1;
            END_IF
          4:
            IF fbFinishHoming.Done THEN
                bHomingInProgress:=FALSE;
                fbFinishHoming.Execute:=FALSE;
                bReadNCVelocities:=FALSE;
                nHomingState:=0;
            END_IF
        END_CASE
   3,4: //Home to bLimitBwd(3) or bLimitFwd(4) using two speeds
        CASE nHomingState OF
          0:
            fbStepLimitSwitchDetection.Execute:=FALSE;
            fbStepLimitSwitchDetection.LimitSwitchMode:=mcRisingEdge;
            fbStepLimitSwitchDetection.Velocity:=fbHomeReadNCVelocities.fVelocityToCam;
            CASE nHomeProcLocal OF
                3: fbStepLimitSwitchDetection.Direction:=mcNegativeDirection;
                4: fbStepLimitSwitchDetection.Direction:=mcPositiveDirection;
            END_CASE
            nHomingState:=nHomingState+1;
          1:
            fbStepLimitSwitchDetection.Execute:=TRUE;
            nHomingState:=nHomingState+1;
          2:
            IF fbStepLimitSwitchDetection.Busy THEN
                nHomingState:=nHomingState+1;
            END_IF
          3:
            IF fbStepLimitSwitchDetection.Done THEN
                fbStepLimitSwitch.Execute:=FALSE;
                fbStepLimitSwitch.LimitSwitchMode:=mcFallingEdge;
                fbStepLimitSwitch.Velocity:=fbHomeReadNCVelocities.fVelocityFromCam;
                fbStepLimitSwitch.Setposition:=fHomePosition;
                CASE nHomeProcLocal OF
                    3: fbStepLimitSwitch.Direction:=mcNegativeDirection;
                    4: fbStepLimitSwitch.Direction:=mcPositiveDirection;
                END_CASE
                nHomingState:=nHomingState+1;
            END_IF
          4:
            fbStepLimitSwitch.Execute:=TRUE;
            nHomingState:=nHomingState+1;
          5:
            IF fbStepLimitSwitch.Busy THEN
                nHomingState:=nHomingState+1;
            END_IF
          6:
            IF fbStepLimitSwitch.Done THEN
                fbFinishHoming.Execute:=TRUE;
                nHomingState:=nHomingState+1;
            END_IF
          7:
            IF fbFinishHoming.Done THEN
                bHomingInProgress:=FALSE;
                fbFinishHoming.Execute:=FALSE;
                bReadNCVelocities:=FALSE;
                nHomingState:=0;
            END_IF
        END_CASE
    11,12: //Home to bHome Sensor moving in the negative(11) or positive(12) direction
        CASE nHomingState OF
          0:
            fbStepAbsoluteSwitch.Execute:=FALSE;
            fbStepAbsoluteSwitch.SwitchMode:=mcRisingEdge;
            fbStepAbsoluteSwitch.SetPosition:=fHomePosition;
            fbStepAbsoluteSwitch.Velocity:=fbHomeReadNCVelocities.fVelocityFromCam;
            CASE nHomeProcLocal OF
                11: fbStepAbsoluteSwitch.Direction:=mcNegativeDirection;
                12: fbStepAbsoluteSwitch.Direction:=mcPositiveDirection;
            END_CASE
            nHomingState:=nHomingState+1;
          1:
            fbStepAbsoluteSwitch.Execute:=TRUE;
            nHomingState:=nHomingState+1;
          2:
            IF fbStepAbsoluteSwitch.Busy THEN
                nHomingState:=nHomingState+1;
            END_IF
          3:
            IF fbStepAbsoluteSwitch.Done THEN
                fbStepAbsoluteSwitch.Execute:=FALSE;
                fbFinishHoming.Execute:=TRUE;
                nHomingState:=nHomingState+1;
            END_IF
          4:
            IF fbFinishHoming.Done THEN
                bHomingInProgress:=FALSE;
                fbFinishHoming.Execute:=FALSE;
                bReadNCVelocities:=FALSE;
                nHomingState:=0;
            END_IF
        END_CASE
    13,14: //Home to bHomeSensor via bLimitBwd(13) or bLimitFwd(14)
        CASE nHomingState OF
          0:
            fbStepLimitSwitchDetection.Execute:=FALSE;
            fbStepLimitSwitchDetection.LimitSwitchMode:=mcRisingEdge;
            fbStepLimitSwitchDetection.Velocity:=fbHomeReadNCVelocities.fVelocityToCam;
            CASE nHomeProcLocal OF
                13: fbStepLimitSwitchDetection.Direction:=mcNegativeDirection;
                14: fbStepLimitSwitchDetection.Direction:=mcPositiveDirection;
            END_CASE
            nHomingState:=nHomingState+1;
          1:
            fbStepLimitSwitchDetection.Execute:=TRUE;
            nHomingState:=nHomingState+1;
          2:
            IF fbStepLimitSwitchDetection.Busy THEN
                nHomingState:=nHomingState+1;
            END_IF
          3:
            IF fbStepLimitSwitchDetection.Done THEN
                fbStepLimitSwitchDetection.Execute:=FALSE;
                CASE nHomeProcLocal OF
                    13: nHomeProcLocal:=12;
                    14: nHomeProcLocal:=11;
                END_CASE
                nHomingState:=0;
            END_IF
        END_CASE
    21,22: //Home to index pulse of an encoder in the negative(21) or positive(22) direction
        CASE nHomingState OF
          0:
            fbStepReferencePulse.Execute:=FALSE;
            fbStepReferencePulse.SetPosition:=fHomePosition;
            fbStepReferencePulse.Velocity:=fbHomeReadNCVelocities.fVelocityFromCam;
            CASE nHomeProcLocal OF
                21: fbStepReferencePulse.Direction:=mcNegativeDirection;
                22: fbStepReferencePulse.Direction:=mcPositiveDirection;
            END_CASE
            nHomingState:=nHomingState+1;
          1:
            fbStepReferencePulse.Execute:=TRUE;
            nHomingState:=nHomingState+1;
          2:
            IF fbStepReferencePulse.Busy THEN
                nHomingState:=nHomingState+1;
            END_IF
          3:
            IF fbStepReferencePulse.Done THEN
                fbStepReferencePulse.Execute:=FALSE;
                fbFinishHoming.Execute:=TRUE;
                nHomingState:=nHomingState+1;
            END_IF
          4:
            IF fbFinishHoming.Done THEN
                bHomingInProgress:=FALSE;
                fbFinishHoming.Execute:=FALSE;
                bReadNCVelocities:=FALSE;
                nHomingState:=0;
            END_IF
        END_CASE
    23,24: //Home to index pulse of an encoder via bLimitBwd(23) or bLimitFwd(24)
        CASE nHomingState OF
          0:
            fbStepLimitSwitchDetection.Execute:=FALSE;
            fbStepLimitSwitchDetection.LimitSwitchMode:=mcRisingEdge;
            fbStepLimitSwitchDetection.Velocity:=fbHomeReadNCVelocities.fVelocityToCam;
            CASE nHomeProcLocal OF
                23: fbStepLimitSwitchDetection.Direction:=mcNegativeDirection;
                24: fbStepLimitSwitchDetection.Direction:=mcPositiveDirection;
            END_CASE
            nHomingState:=nHomingState+1;
          1:
            fbStepLimitSwitchDetection.Execute:=TRUE;
            nHomingState:=nHomingState+1;
          2:
            IF fbStepLimitSwitchDetection.Busy THEN
                nHomingState:=nHomingState+1;
            END_IF
          3:
            IF fbStepLimitSwitchDetection.Done THEN
                fbStepLimitSwitchDetection.Execute:=FALSE;
                CASE nHomeProcLocal OF
                    23: nHomeProcLocal:=22;
                    24: nHomeProcLocal:=21;
                END_CASE
                nHomingState:=0;
            END_IF
        END_CASE
    90: //Set current position without moving
       CASE nHomingState OF
          0:
            fbHomeDirect.Execute:=FALSE;
            fbHomeDirect.SetPosition:=fHomePosition;
            nHomingState:=nHomingState+1;
          1:
            fbHomeDirect.Execute:=TRUE;
            nHomingState:=nHomingState+1;
          2: // Check that started
            IF fbHomeDirect.Busy THEN
                nHomingState:=nHomingState+1;
            END_IF
          3: // Check that finished
            IF fbHomeDirect.Done THEN
                fbHomeDirect.Execute:=FALSE;
                bHomingInProgress:=FALSE;
                bReadNCVelocities:=FALSE;
                nHomingState:=0;
            END_IF
        END_CASE
END_CASE
ELSE
    fbStepLimitSwitch.Execute:=FALSE;
    fbStepLimitSwitchDetection.Execute:=FALSE;
    fbStepAbsoluteSwitch.Execute:=FALSE;
    fbStepReferencePulse.Execute:=FALSE;
    fbHomeDirect.Execute:=FALSE;
    nHomingState:=0;
END_IF

fbHomeReadNCVelocities(
    En:=TRUE,
    bExecute:=bReadNCVelocities,
    bReset:=bReset,
    Axis:=Axis );

StOptions2.DisableDriveAccess:=TRUE;
StOptions4.DisableDriveAccess:=TRUE;
stOptions4.EnableLagErrorDetection:=TRUE;

IF fbStepLimitSwitch.Direction=mcPositiveDirection THEN
    fbRef_Signal_Ref1.Level:=NOT(bLimitFwd);
ELSIF fbStepLimitSwitch.Direction=mcNegativeDirection THEN
    fbRef_Signal_Ref1.Level:=NOT(bLimitBwd);
END_IF
fbStepLimitSwitch(
    Axis:= Axis,
    Parameter:= fbHomingParameter,
    LimitSwitchSignal:= fbRef_Signal_Ref1,
    Options:= StOptions4);

IF fbStepLimitSwitchDetection.Direction=mcPositiveDirection THEN
    fbRef_Signal_Ref2.Level:=NOT(bLimitFwd);
ELSIF fbStepLimitSwitchDetection.Direction=mcNegativeDirection THEN
    fbRef_Signal_Ref2.Level:=NOT(bLimitBwd);
END_IF
fbStepLimitSwitchDetection(
    Axis:= AXIS,
    Parameter:= fbHomingParameter,
    Execute:= ,
    Direction:= ,
    LimitSwitchMode:= ,
    LimitSwitchSignal:= fbRef_Signal_Ref2,
    TimeLimit:= tLimit,
    Options:= StOptions4);

fbRef_Signal_Ref3.Level:=bHomeSensor;
fbRef_Signal_Ref3.TouchProbe:=PlcEvent;
fbRef_Signal_Ref3.SignalSource:=SignalSource_Default;
fbStepAbsoluteSwitch(
    Axis:= Axis,
    Parameter:= fbHomingParameter,
    ReferenceSignal:= fbRef_Signal_Ref3,
    TimeLimit:= tLimit,
    PositiveLimitSwitch:=NOT(bLimitFwd),
    NegativeLimitSwitch:=NOT(bLimitBwd),
    Options:= StOptions4);

fbRef_Signal_Ref4.SignalSource:=SignalSource_ZeroPulse;
fbRef_Signal_Ref4.TouchProbe:=TouchProbe1;
fbStepReferencePulse(
    Axis:= Axis,
    Parameter:= fbHomingParameter,
    ReferenceSignal:= fbRef_Signal_Ref4,
    TimeLimit:= tLimit,
    Options:= StOptions4);

fbHomeDirect(
    Axis:= Axis,
    Parameter:= fbHomingParameter,
    Options:= StOptions2);

fbFinishHoming(
    Axis:= Axis,
    Parameter:= fbHomingParameter,
    Velocity:=,
    Options:= StOptions2);

fbAbortHoming(
    Axis:= Axis,
    Parameter:= fbHomingParameter,
    Options:= StOptions2);

IF fbStepLimitSwitch.Error THEN
    bError:=TRUE;
    nErrorId:=fbStepLimitSwitch.ErrorID;
ELSIF fbStepLimitSwitchDetection.Error THEN
    bError:=TRUE;
    nErrorId:=fbStepLimitSwitchDetection.ErrorID;
ELSIF fbStepAbsoluteSwitch.Error THEN
    bError:=TRUE;
    nErrorId:=fbStepAbsoluteSwitch.ErrorID;
ELSIF fbStepReferencePulse.Error THEN
    bError:=TRUE;
    nErrorId:=fbStepReferencePulse.ErrorID;
ELSIF fbHomeDirect.Error THEN
    bError:=TRUE;
    nErrorId:=fbHomeDirect.ErrorID;
ELSIF fbAbortHoming.Error THEN
    bError:=TRUE;
    nErrorId:=fbAbortHoming.ErrorID;
ELSIF fbFinishHoming.Error THEN
    bError:=TRUE;
    nErrorId:=fbFinishHoming.ErrorID;
END_IF

IF fbStepLimitSwitch.CommandAborted OR fbStepLimitSwitchDetection.CommandAborted OR fbStepAbsoluteSwitch.CommandAborted OR fbStepReferencePulse.CommandAborted OR fbHomeDirect.CommandAborted THEN
    nHomingState:=0;
    bHomingInProgress:=FALSE;
    bWarning:=TRUE;
END_IF

bHomed:=Axis.Status.Homed;

END_FUNCTION_BLOCK

// ---- tc_mca_std_lib/POUs/Motion/Homing/FB_HomeReadNcVelocities.TcPOU
FUNCTION_BLOCK FB_HomeReadNcVelocities
VAR_INPUT
    En: BOOL;
    bReset: BOOL;
    bExecute: BOOL;
END_VAR
VAR_IN_OUT
    Axis: AXIS_REF;
END_VAR
VAR_OUTPUT
    EnO: BOOL;
    bBusy: BOOL;
    bDone: BOOL;
    bError: BOOL;
    nErrorId: UDINT;
    fVelocityToCam: LREAL;
    fVelocityFromCam: LREAL;
END_VAR
VAR
    fbReadVelocityToCam:FB_ReadFloatParameter;
    fbReadVelocityFromCam:FB_ReadFloatParameter;
END_VAR

En:=EnO;
IF bReset THEN
    bError:=FALSE;
    nErrorId:=0;
END_IF

fbReadVelocityToCam(
    bExecute:=bExecute,
    nDeviceGroup:= 16#4000,
    nIndexOffset:= 16#6,
    Axis:= Axis);

fbReadVelocityFromCam(
    bExecute:=bExecute,
    nDeviceGroup:= 16#4000,
    nIndexOffset:= 16#7,
    Axis:= Axis);

fVelocityToCam:=fbReadVelocityToCam.nData;
fVelocityFromCam:=fbReadVelocityFromCam.nData;

bBusy:=fbReadVelocityFromCam.bBusy OR fbReadVelocityToCam.bBusy;
bDone:=fbReadVelocityFromCam.bDone AND fbReadVelocityToCam.bDone AND bExecute;

bError:=fbReadVelocityToCam.bError OR fbReadVelocityFromCam.bError;
IF fbReadVelocityToCam.bError THEN
  nErrorId:=fbReadVelocityToCam.nErrorId;
ELSIF fbReadVelocityFromCam.bError THEN
  nErrorId:=fbReadVelocityFromCam.nErrorId;
END_IF

END_FUNCTION_BLOCK

// ---- tc_mca_std_lib/POUs/ChangeConfig/FB_ReadFloatParameter.TcPOU
FUNCTION_BLOCK FB_ReadFloatParameter
VAR_INPUT
    bExecute: BOOL;
    ///16#4000=Axisdata, 16#5000=Encoderdata, 16#6000=Controldata, 16#7000=Drivedata
    nDeviceGroup: UDINT;
    nIndexOffset: UDINT;
END_VAR
VAR_OUTPUT
    nData: LREAL;
    bBusy: BOOL;
    bDone: BOOL;
    bError: BOOL;
    nErrorId: UDINT;
END_VAR
VAR_IN_OUT
    Axis: AXIS_REF;
END_VAR
VAR
    nState: UINT;
    fbADSREAD: ADSREAD;
END_VAR

(*Sequence to read parameter in Nc*)
CASE nState OF
0:  (*Start sequence. Wait until bExecute is TRUE*)
    IF bExecute THEN
        bBusy:=TRUE;
        bError:=FALSE;
        nErrorId:=0;
        nState:=10;
    END_IF

10: (*Read parameter in Nc*)
    fbADSREAD(
        PORT:=500,
        IDXGRP:=nDeviceGroup+Axis.NcToPlc.AxisId,
        IDXOFFS:=nIndexOffset,
        LEN:=SIZEOF(nData),
        DESTADDR:=ADR(nData),
        READ:=TRUE);

    (*Wait until it's done or if an error occurs*)
    IF NOT fbADSREAD.ERR THEN
        IF NOT fbADSREAD.BUSY THEN
            fbADSREAD(READ:=FALSE);
            nState:=20;
        END_IF
    ELSE
        nErrorId:=fbADSREAD.ERRID;
        nState:=999;
    END_IF

20: (*Sequense is done. Waits until bExecute is FALSE*)
    bBusy:=FALSE;
    bDone:=TRUE;
    IF NOT bExecute THEN
        bDone:=FALSE;
        nState:=0;
    END_IF

999: (*Error in sequence*)
    bError:=TRUE;
    bBusy:=FALSE;
    bDone:=FALSE;
    fbADSREAD(READ:=FALSE);
    IF NOT bExecute THEN
        nState:=0;
    END_IF

END_CASE

END_FUNCTION_BLOCK

// ---- tc_mca_std_lib/POUs/ErrorHandling/FB_ErrorSystem.TcPOU
FUNCTION_BLOCK FB_ErrorSystem

VAR_INPUT
    En                  : BOOL;                         //Enable input
    bReset              : BOOL;                         //Delete all Error entry
    nErrorNum           : ULINT;                        //ErrorID to be acknoledged
    bACK                : BOOL;                         //Acknoledge the given error and delete it from the list
    bValidSelection     : BOOL;                         //Visu table valid selection flag
    nTableRowIndex      : INT;                          //Visu table selected row index
END_VAR

VAR_OUTPUT
    EnO                 : BOOL;                         //Enable output
    nSelectedError      : ULINT;                        //Currently selected errorID
    pErrorSystem        : POINTER TO ST_ErrorSystem;    //Pointer to ErrorSystem
END_VAR

VAR_IN_OUT

END_VAR

VAR
    nFreePos : UINT;                                    //Number of free position in the list
    nListCnt1 : UINT;                                   //work variable
    ErrorSystem : ST_ErrorSystem;                       //Data structure of the Error list

    bAckInternal        : BOOL;
    bResetInternal      : BOOL;
    nErrorNumInternal   : ULINT;

    Ack_trig        : R_TRIG;
    RST_trig        : R_TRIG;
    nNoErrorPrev    : UINT;
    nNoActivePrev   : UINT;
    nErrorNumPrev   : ULINT;
END_VAR

(*
* ================================================================================
*                                   DESCRIPTION
* ================================================================================
* This Function Block implements the core structure of the Error/Warning Handling
* system. It realizes the datastructure containing every Error Entry, collect
* statistics about the usage and manage the Error Entries.
* ================================================================================
*)
EnO := En;

//Ponter to ErrorSystem
pErrorSystem := ADR(ErrorSystem);

//Rising-edge detection on inputs
Ack_trig (
    CLK     := bAck,
    Q       => bAckInternal,
);

RST_trig (
    CLK     := bReset,
    Q       => bResetInternal,
);

//Entry selection decision
IF bValidSelection AND nErrorNum = 0 THEN
    nErrorNumInternal := ErrorSystem.aErrorData[nTableRowIndex].ErrorNum;
ELSE
    nErrorNumInternal := nErrorNum;
END_IF

nSelectedError := nErrorNumInternal;

//Reset the system
IF bResetInternal THEN
    MEMSET ( ADR(ErrorSystem.aErrorData[0]), 0, cSizeOfErrorData * SIZEOF(ST_ErrorEntry));
    ErrorSystem.nNextErrorNum := 1;
END_IF

//Number of errors
ErrorSystem.nNoError := 0;
ErrorSystem.nNoActive := 0;
ErrorSystem.nNoInactive := 0;
FOR nListCnt1 := 0 TO cSizeOfErrorData - 1 DO
    IF ErrorSystem.aErrorData[nListCnt1].ErrorNum <> 0  THEN
        ErrorSystem.nNoError := ErrorSystem.nNoError+1;
        IF ErrorSystem.aErrorData[nListCnt1].ErrorState = DUT_ErrorState.Active THEN
            ErrorSystem.nNoActive := ErrorSystem.nNoActive + 1;
        ELSE
            ErrorSystem.nNoInactive := ErrorSystem.nNoInactive + 1;
        END_IF
    END_IF
END_FOR

//Number of free positions
nFreePos := cSizeOfErrorData - ErrorSystem.nNoError;

//Acknoledge specified Error entry
IF bAckInternal THEN
    FOR nListCnt1 := 0 TO cSizeOfErrorData - 1 DO
        IF ErrorSystem.aErrorData[nListCnt1].ErrorNum = nErrorNumInternal THEN
            ErrorSystem.aErrorData[nListCnt1].ErrorState := DUT_ErrorState.Acknowledged;
        END_IF
    END_FOR
END_IF

//Deleting acknoledged errors
FOR nListCnt1 := 0 TO cSizeOfErrorData - 1 DO
    IF ErrorSystem.aErrorData[nListCnt1].ErrorState = DUT_ErrorState.Acknowledged THEN
        MEMMOVE (ADR(ErrorSystem.aErrorData[nListCnt1]), ADR(ErrorSystem.aErrorData[nListCnt1+1]), (cSizeOfErrorData - 1 - nListCnt1) * SIZEOF(ST_ErrorEntry));
        MEMSET(ADR(ErrorSystem.aErrorData[cSizeOfErrorData - 1]), 0, SIZEOF(ST_ErrorEntry));
    END_IF
END_FOR

IF ErrorSystem.nNoError <> nNoErrorPrev OR ErrorSystem.nNoActive <> nNoActivePrev  THEN
    nNoErrorPrev    := ErrorSystem.nNoError;
    nNoActivePrev   := ErrorSystem.nNoActive;
    //Copy the structure to GVL
    MEMCPY ( ADR(GVL.stErrorSystemCom), ADR(ErrorSystem), SIZEOF(ST_ErrorSystem));
END_IF

END_FUNCTION_BLOCK

// ---- tc_mca_std_lib/POUs/ErrorHandling/FB_NC_Error.TcPOU
FUNCTION_BLOCK FB_NC_Error

VAR_INPUT
    En              : BOOL;
    nNC_ErrorID     : UDINT;
    nNC_AxisID      : UDINT;
    ErrorSystem     : POINTER TO ST_ErrorSystem;
END_VAR

VAR_OUTPUT
    EnO         : BOOL;
    bError      : BOOL;
END_VAR

VAR
    NCError             : FB_GenericError;
END_VAR

(*
* ================================================================================
*                                   DESCRIPTION
* ================================================================================
* This Function Block connects FB_DriveVirtual's error output to the Error System.
* Link the corresponding outputs of FB_DriveVirtual to the inputs of this FB.
* ================================================================================
*)

IF En THEN
    EnO := En;

    IF nNC_ErrorID <> 0 THEN
        NCError.sErrorMessage   := 'Axis ';
        NCError.sErrorMessage   := CONCAT (NCError.sErrorMessage, UDINT_TO_STRING(nNC_AxisID));
        NCError.sErrorMessage   := CONCAT (NCError.sErrorMessage, ' is in error state. NC error ID (Hex): 0x');
        NCError.sErrorMessage   := CONCAT (NCError.sErrorMessage, DWORD_TO_HEXSTR(nNC_ErrorID,4,FALSE));
        NCError.ErrorPriority   := 6;
        NCError.bError          := TRUE;
    ELSE
        NCError.sErrorMessage   := '';
        NCError.bError          := FALSE;
        NCError.ErrorPriority   := 0;
    END_IF

END_IF

NCError (
    En                  := TRUE,
    bError              := ,
    sErrorMessage       := ,
    ErrorPriority       := ,
    iTerminal_ID        := ,
    pErrorSystem        := ErrorSystem,
    EnO     => ,
);


(*
        NCError.sErrorMessage := CONCAT (NCError.sErrorMessage, ': ');
        CASE nNC_ErrorID OF
            //General NC Errors
            16#4000 :   NCError.sErrorMessage := CONCAT (NCError.sErrorMessage,     'Internal Error; ');
            16#4001 :   NCError.sErrorMessage := CONCAT (NCError.sErrorMessage,     'Memory Error; ');
            16#4002 :   NCError.sErrorMessage := CONCAT (NCError.sErrorMessage,     'NC retain data error (persistent data); ');
            16#4010 :   NCError.sErrorMessage := CONCAT (NCError.sErrorMessage,     'Channel identifier not allowed; ');
            16#4011 :   NCError.sErrorMessage := CONCAT (NCError.sErrorMessage,     'Group identifier not allowed; ');
            16#4012 :   NCError.sErrorMessage := CONCAT (NCError.sErrorMessage,     'Axis identifier not allowed; ');
            16#4013 :   NCError.sErrorMessage := CONCAT (NCError.sErrorMessage,     'Encoder identifier not allowed; ');
            16#4014 :   NCError.sErrorMessage := CONCAT (NCError.sErrorMessage,     'Controller identifier not allowed; ');
            16#4015 :   NCError.sErrorMessage := CONCAT (NCError.sErrorMessage,     'Drive identifier not allowed; ');
            16#4016 :   NCError.sErrorMessage := CONCAT (NCError.sErrorMessage,     'Table identifier not allowed; ');
            16#4020 :   NCError.sErrorMessage := CONCAT (NCError.sErrorMessage,     'No process image; ');
            16#4021 :   NCError.sErrorMessage := CONCAT (NCError.sErrorMessage,     'No process image; ');
            16#4022 :   NCError.sErrorMessage := CONCAT (NCError.sErrorMessage,     'No process image; ');
            16#4023 :   NCError.sErrorMessage := CONCAT (NCError.sErrorMessage,     'No process image; ');
            16#4024 :   NCError.sErrorMessage := CONCAT (NCError.sErrorMessage,     'No process image; ');
            16#4025 :   NCError.sErrorMessage := CONCAT (NCError.sErrorMessage,     'No process image; ');
            16#4030 :   NCError.sErrorMessage := CONCAT (NCError.sErrorMessage,     'Coupling type not allowed; ');
            16#4031 :   NCError.sErrorMessage := CONCAT (NCError.sErrorMessage,     'Axis type not allowed; ');
            16#4040 :   NCError.sErrorMessage := CONCAT (NCError.sErrorMessage,     'Axis is incompatible; ');
            16#4050 :   NCError.sErrorMessage := CONCAT (NCError.sErrorMessage,     'Channel not ready for operation; ');
            16#4051 :   NCError.sErrorMessage := CONCAT (NCError.sErrorMessage,     'Group not ready for operation; ');
            16#4052 :   NCError.sErrorMessage := CONCAT (NCError.sErrorMessage,     'Axis not ready for operation; ');
            16#4060 :   NCError.sErrorMessage := CONCAT (NCError.sErrorMessage,     'Channel exists; ');
            16#4061 :   NCError.sErrorMessage := CONCAT (NCError.sErrorMessage,     'Group exists; ');
            16#4062 :   NCError.sErrorMessage := CONCAT (NCError.sErrorMessage,     'Axis exists; ');
            16#4063 :   NCError.sErrorMessage := CONCAT (NCError.sErrorMessage,     'Table exists; ');
            16#4070 :   NCError.sErrorMessage := CONCAT (NCError.sErrorMessage,     'Axis index not allowed; ');
            16#4071 :   NCError.sErrorMessage := CONCAT (NCError.sErrorMessage,     'Axis index not allowed; ');

            //Channel Errors
            16#4101 :   NCError.sErrorMessage := CONCAT (NCError.sErrorMessage,     'Group index not allowed; ');
            16#4102 :   NCError.sErrorMessage := CONCAT (NCError.sErrorMessage,     'Null pointer; ');
            16#4103 :   NCError.sErrorMessage := CONCAT (NCError.sErrorMessage,     'No process image; ');
            16#4104 :   NCError.sErrorMessage := CONCAT (NCError.sErrorMessage,     'M-function index not allowed; ');
            16#4105 :   NCError.sErrorMessage := CONCAT (NCError.sErrorMessage,     'No memmory; ');
            16#4106 :   NCError.sErrorMessage := CONCAT (NCError.sErrorMessage,     'Not ready; ');
            16#4107 :   NCError.sErrorMessage := CONCAT (NCError.sErrorMessage,     'Function/command not supported; ');
            16#4108 :   NCError.sErrorMessage := CONCAT (NCError.sErrorMessage,     'Invalid parameter while starting; ');
            16#4109 :   NCError.sErrorMessage := CONCAT (NCError.sErrorMessage,     'Channel function/command not executable; ');
            16#410A :   NCError.sErrorMessage := CONCAT (NCError.sErrorMessage,     'ItpGoAhead not executable; ');
            16#4110 :   NCError.sErrorMessage := CONCAT (NCError.sErrorMessage,     'Error opening a file; ');
            16#4111 :   NCError.sErrorMessage := CONCAT (NCError.sErrorMessage,     'Syntax error during loading; ');
            16#4112 :   NCError.sErrorMessage := CONCAT (NCError.sErrorMessage,     'Syntax error  during interpretation; ');
            16#4113 :   NCError.sErrorMessage := CONCAT (NCError.sErrorMessage,     'Missing subroutine; ');
            16#4114 :   NCError.sErrorMessage := CONCAT (NCError.sErrorMessage,     'Loading buffer of interpreter is too small; ');
            16#4117 :   NCError.sErrorMessage := CONCAT (NCError.sErrorMessage,     'Subroutine incomplete; ');
            16#4118 :   NCError.sErrorMessage := CONCAT (NCError.sErrorMessage,     'Error while loading the NC program; ');
            16#4119 :   NCError.sErrorMessage := CONCAT (NCError.sErrorMessage,     'Error while loading the NC program; ');
            16#4120 :   NCError.sErrorMessage := CONCAT (NCError.sErrorMessage,     'Devide by zero; ');
            16#4121 :   NCError.sErrorMessage := CONCAT (NCError.sErrorMessage,     'Invalide circle parameterization; ');
            16#4122 :   NCError.sErrorMessage := CONCAT (NCError.sErrorMessage,     'Invalid FPU-Operation; ');
            16#4130 :   NCError.sErrorMessage := CONCAT (NCError.sErrorMessage,     'Stack overflow: subroutines; ');
            16#4131 :   NCError.sErrorMessage := CONCAT (NCError.sErrorMessage,     'Stack underflow: subroutines; ');
            16#4132 :   NCError.sErrorMessage := CONCAT (NCError.sErrorMessage,     'Stack overflow: arithmetic unit; ');
            16#4133 :   NCError.sErrorMessage := CONCAT (NCError.sErrorMessage,     'Stack underflow: arithmetic unit; ');
            16#4140 :   NCError.sErrorMessage := CONCAT (NCError.sErrorMessage,     'Register index not allowed; ');
            16#4141 :   NCError.sErrorMessage := CONCAT (NCError.sErrorMessage,     'Unaccaptable G-function index; ');
            16#4142 :   NCError.sErrorMessage := CONCAT (NCError.sErrorMessage,     'Unaccaptable M-function index; ');
            16#4143 :   NCError.sErrorMessage := CONCAT (NCError.sErrorMessage,     'Unacceptable extended address; ');
            16#4144 :   NCError.sErrorMessage := CONCAT (NCError.sErrorMessage,     'Unaccaptable index of internal H-function; ');
            16#4145 :   NCError.sErrorMessage := CONCAT (NCError.sErrorMessage,     'Machine data value unacceptable; ');
            16#4150 :   NCError.sErrorMessage := CONCAT (NCError.sErrorMessage,     'Cannot change tool params here; ');
            16#4151 :   NCError.sErrorMessage := CONCAT (NCError.sErrorMessage,     'Cannoot calculate tool compensation; ');
            16#4152 :   NCError.sErrorMessage := CONCAT (NCError.sErrorMessage,     'Tool compensation; ');
            16#4153 :   NCError.sErrorMessage := CONCAT (NCError.sErrorMessage,     'Tool compensation; ');
            16#4153 :   NCError.sErrorMessage := CONCAT (NCError.sErrorMessage,     'Tool compensation; ');


        END_CASE
*)

END_FUNCTION_BLOCK

// ---- tc_mca_std_lib/POUs/ErrorHandling/FB_GenericError.TcPOU
FUNCTION_BLOCK FB_GenericError

//Inputs
VAR_INPUT
    En                  : BOOL;
    bError              : BOOL;
    sErrorMessage       : STRING;
    ErrorPriority       : INT;
    iTerminal_ID        : INT;
    pErrorSystem        : POINTER TO ST_ErrorSystem;
END_VAR

//Outputs
VAR_OUTPUT
    EnO             : BOOL;
END_VAR


VAR
    LocalEntry          : ST_ErrorEntry;
    //
    sMessagePrev        : STRING;
    bMsgChanged         : BOOL;
    nErrSysCNT          :UINT;

END_VAR

(*
* ================================================================================
*                                   DESCRIPTION
* ================================================================================
* This Function Block creates a generic connection to the Error System. Unlike
* FB_TerminalError, this does not evaluate variables. Instead it checks the
* sErrorMessage & bError input variables. If bError becomes '1', a new entry is
* created in the Error System. As long as bError stays '1' every change in
* sErrorMessage inactivate the previous Error and creates a new one with the new
* message. When bError becomes '0' the last enrty is set to inactive.
* ================================================================================
*)

//Connect En to EnO
EnO := En;

IF En THEN
    //Check if pointer is OK
    IF pErrorSystem=0 THEN RETURN; END_IF

    IF sErrorMessage <> sMessagePrev THEN
        bMsgChanged := TRUE;
    ELSE
        bMsgChanged := FALSE;
    END_IF

    //Update previous value
    sMessagePrev := sErrorMessage;

    IF bMsgChanged THEN
        IF bError THEN
            IF LocalEntry.ErrorState = DUT_ErrorState.Active THEN       //Close active error
                //Read system time
                LocalEntry.sDateTimeOff := Tc2_EtherCat.DCTIME64_TO_STRING(Tc2_EtherCAT.F_GetActualDcTime64());
                LocalEntry.ErrorState   := DUT_ErrorState.Inactive;
                //Write Off-time to Error System
                FOR nErrSysCNT := 0 TO cSizeOfErrorData - 1 DO
                    IF pErrorSystem^.aErrorData[nErrSysCNT].ErrorNum = LocalEntry.ErrorNum THEN
                        pErrorSystem^.aErrorData[nErrSysCNT].sDateTimeOff   := LocalEntry.sDateTimeOff;
                        pErrorSystem^.aErrorData[nErrSysCNT].ErrorState     := DUT_ErrorState.Inactive;
                        EXIT;
                    END_IF
                END_FOR

                //Clear ErrorData
                MEMSET(ADR(LocalEntry), 0, SIZEOF(LocalEntry));
            END_IF

            //Open a new error
            LocalEntry.ErrorState       := DUT_ErrorState.Active;                                               //Set Error State
            LocalEntry.sDateTimeOn      := Tc2_EtherCat.DCTIME64_TO_STRING(Tc2_EtherCAT.F_GetActualDcTime64()); //Convert to string
            LocalEntry.sErrorMessage    := sErrorMessage;                                                       //Write message into the entry
            LocalEntry.ErrorPriority    := ErrorPriority;                                                       //Priority
            LocalEntry.iTerminalID      := iTerminal_ID;                                                        //Terminal_ID

            //Check for overflow
            IF pErrorSystem^.nNoError >= cSizeOfErrorData THEN
                pErrorSystem^.nNoOverflow   := pErrorSystem^.nNoOverflow+1;
            END_IF

            //Write Error Data into Error System
            LocalEntry.ErrorNum := pErrorSystem^.nNExtErrorNum ;
            MEMMOVE( ADR(pErrorSystem^.aErrorData[1]), ADR(pErrorSystem^.aErrorData[0]), (cSizeOfErrorData-1) * SIZEOF(ST_ErrorEntry));
            pErrorSystem^.aErrorData[0] := LocalEntry;
            pErrorSystem^.nNExtErrorNum := pErrorSystem^.nNExtErrorNum+1;

        ELSE
            //Close Active Error
            //Read system time
            LocalEntry.sDateTimeOff := Tc2_EtherCat.DCTIME64_TO_STRING(Tc2_EtherCAT.F_GetActualDcTime64());
            LocalEntry.ErrorState   := DUT_ErrorState.Inactive;

            //Write Off time to Error System
            FOR nErrSysCNT := 0 TO cSizeOfErrorData - 1 DO
                IF pErrorSystem^.aErrorData[nErrSysCNT].ErrorNum = LocalEntry.ErrorNum THEN
                    pErrorSystem^.aErrorData[nErrSysCNT].sDateTimeOff   := LocalEntry.sDateTimeOff;
                    pErrorSystem^.aErrorData[nErrSysCNT].ErrorState     := LocalEntry.ErrorState;
                    EXIT;
                END_IF
            END_FOR

            //Clear ErrorData
            MEMSET(ADR(LocalEntry), 0, SIZEOF(LocalEntry));
        END_IF
    END_IF

END_IF

END_FUNCTION_BLOCK

// ---- tc_mca_std_lib/POUs/ChangeConfig/FB_ReadParameterInNc_v1_00.TcPOU
///#########################################################
///Function block to read parameter in Nc.
///
/// Library:
/// Tc2_MC2.lib
/// Tc2_System.lib
///
/// Global Variables:
///
/// Data types:
///
/// External functions:
///
/// History:
/// 2014-02-05  v1.00   NB  Release code.
///
/// Known bugs:
///
///
///
///###########################################################
FUNCTION_BLOCK FB_ReadParameterInNc_v1_00
VAR_INPUT
    bExecute: BOOL;
    ///16#4000=Axisdata, 16#5000=Encoderdata, 16#6000=Controldata, 16#7000=Drivedata
    nDeviceGroup: UDINT;
    nIndexOffset: UDINT;
END_VAR
VAR_OUTPUT
    nData: DWORD;
    bBusy: BOOL;
    bDone: BOOL;
    bError: BOOL;
    nErrorId: UDINT;
END_VAR
VAR_IN_OUT
    Axis: AXIS_REF;
END_VAR
VAR
    nState: UINT;
    fbADSREAD: ADSREAD;
END_VAR

(*Sequence to read parameter in Nc*)
CASE nState OF
0:  (*Start sequence. Wait until bExecute is TRUE*)
    IF bExecute THEN
        bBusy:=TRUE;
        bError:=FALSE;
        nErrorId:=0;
        nState:=10;
    END_IF

10: (*Read parameter in Nc*)
    fbADSREAD(
        PORT:=500,
        IDXGRP:=nDeviceGroup+Axis.NcToPlc.AxisId,
        IDXOFFS:=nIndexOffset,
        LEN:=SIZEOF(nData),
        DESTADDR:=ADR(nData),
        READ:=TRUE);

    (*Wait until it's done or if an error occurs*)
    IF NOT fbADSREAD.ERR THEN
        IF NOT fbADSREAD.BUSY THEN
            fbADSREAD(READ:=FALSE);
            nState:=20;
        END_IF
    ELSE
        nErrorId:=fbADSREAD.ERRID;
        nState:=999;
    END_IF

20: (*Sequense is done. Waits until bExecute is FALSE*)
    bBusy:=FALSE;
    bDone:=TRUE;
    IF NOT bExecute THEN
        bDone:=FALSE;
        nState:=0;
    END_IF

999: (*Error in sequence*)
    bError:=TRUE;
    bBusy:=FALSE;
    bDone:=FALSE;
    fbADSREAD(READ:=FALSE);
    IF NOT bExecute THEN
        nState:=0;
    END_IF

END_CASE

END_FUNCTION_BLOCK

// ---- tc_mca_std_lib/POUs/ChangeConfig/FB_WriteFloatParameter.TcPOU
///#########################################################
///Function block to write parameter in Nc.
///
/// Library:
/// Tc2_MC2.lib
/// Tc2_System.lib
///
/// Global Variables:
///
/// Data types:
///
/// External functions:
///
/// History:
/// 2014-02-05  v1.00   NB  Release code.
///
/// Known bugs:
///
///
///
///###########################################################
FUNCTION_BLOCK FB_WriteFloatParameter
VAR_INPUT
    bExecute: BOOL;
    ///16#4000=Axisdata, 16#5000=Encoderdata, 16#6000=Controldata, 16#7000=Drivedata
    nDeviceGroup: UDINT;
    nIndexOffset: UDINT;
    nData: LREAL;
END_VAR
VAR_OUTPUT
    bBusy: BOOL;
    bDone: BOOL;
    bError: BOOL;
    nErrorId: UDINT;
END_VAR
VAR_IN_OUT
    Axis: AXIS_REF;
END_VAR
VAR
    nState: UINT;
    fbADSWRITE: ADSWRITE;
END_VAR

(*Sequence to write parameter in Nc*)
CASE nState OF
0:  (*Start sequence. Wait until bExecute is TRUE*)
    IF bExecute THEN
        bBusy:=TRUE;
        bError:=FALSE;
        nErrorId:=0;
        nState:=10;
    END_IF

10: (*Write parameter in Nc*)
    fbADSWRITE(
        PORT:=500,
        IDXGRP:=nDeviceGroup+Axis.NcToPlc.AxisId,
        IDXOFFS:=nIndexOffset,
        LEN:=SIZEOF(nData),
        SRCADDR:=ADR(nData),
        WRITE:=TRUE);

    (*Wait until it's done or if an error occurs*)
    IF NOT fbADSWRITE.ERR THEN
        IF NOT fbADSWRITE.BUSY THEN
            fbADSWRITE(WRITE:=FALSE);
            nState:=20;
        END_IF
    ELSE
        nErrorId:=fbADSWRITE.ERRID;
        nState:=999;
    END_IF

20: (*Sequense is done. Waits until bExecute is FALSE*)
    bBusy:=FALSE;
    bDone:=TRUE;
    IF NOT bExecute THEN
        bDone:=FALSE;
        nState:=0;
    END_IF

999: (*Error in sequence*)
    bError:=TRUE;
    bBusy:=FALSE;
    bDone:=FALSE;
    fbADSWRITE(WRITE:=FALSE);
    IF NOT bExecute THEN
        nState:=0;
    END_IF

END_CASE

END_FUNCTION_BLOCK

// ---- tc_mca_std_lib/POUs/ChangeConfig/FB_WriteParameterInNc_v1_00.TcPOU
///#########################################################
///Function block to write parameter in Nc.
///
/// Library:
/// Tc2_MC2.lib
/// Tc2_System.lib
///
/// Global Variables:
///
/// Data types:
///
/// External functions:
///
/// History:
/// 2014-02-05  v1.00   NB  Release code.
///
/// Known bugs:
///
///
///
///###########################################################
FUNCTION_BLOCK FB_WriteParameterInNc_v1_00
VAR_INPUT
    bExecute: BOOL;
    ///16#4000=Axisdata, 16#5000=Encoderdata, 16#6000=Controldata, 16#7000=Drivedata
    nDeviceGroup: UDINT;
    nIndexOffset: UDINT;
    nData: DWORD;
END_VAR
VAR_OUTPUT
    bBusy: BOOL;
    bDone: BOOL;
    bError: BOOL;
    nErrorId: UDINT;
END_VAR
VAR_IN_OUT
    Axis: AXIS_REF;
END_VAR
VAR
    nState: UINT;
    fbADSWRITE: ADSWRITE;
END_VAR

(*Sequence to write parameter in Nc*)
CASE nState OF
0:  (*Start sequence. Wait until bExecute is TRUE*)
    IF bExecute THEN
        bBusy:=TRUE;
        bError:=FALSE;
        nErrorId:=0;
        nState:=10;
    END_IF

10: (*Write parameter in Nc*)
    fbADSWRITE(
        PORT:=500,
        IDXGRP:=nDeviceGroup+Axis.NcToPlc.AxisId,
        IDXOFFS:=nIndexOffset,
        LEN:=SIZEOF(nData),
        SRCADDR:=ADR(nData),
        WRITE:=TRUE);

    (*Wait until it's done or if an error occurs*)
    IF NOT fbADSWRITE.ERR THEN
        IF NOT fbADSWRITE.BUSY THEN
            fbADSWRITE(WRITE:=FALSE);
            nState:=20;
        END_IF
    ELSE
        nErrorId:=fbADSWRITE.ERRID;
        nState:=999;
    END_IF

20: (*Sequense is done. Waits until bExecute is FALSE*)
    bBusy:=FALSE;
    bDone:=TRUE;
    IF NOT bExecute THEN
        bDone:=FALSE;
        nState:=0;
    END_IF

999: (*Error in sequence*)
    bError:=TRUE;
    bBusy:=FALSE;
    bDone:=FALSE;
    fbADSWRITE(WRITE:=FALSE);
    IF NOT bExecute THEN
        nState:=0;
    END_IF

END_CASE

END_FUNCTION_BLOCK

// ---- tc_mca_std_lib/POUs/ErrorHandling/FB_TerminalError.TcPOU
FUNCTION_BLOCK FB_TerminalError

VAR_INPUT
    En                  : BOOL;
    iTerminal_ID        : INT;
    bWcState            : BOOL;
    uiInfoData_State    : UINT;
    pErrorSystem        : POINTER TO ST_ErrorSystem;                    //Pointer to the error system
END_VAR

VAR_OUTPUT
    EnO : BOOL;
    bError : BOOL := FALSE;
END_VAR

VAR
    iStateError : UINT;
    iOtherError : UINT;
    ErrorData   : ST_ErrorEntry;
    nErrSysCNT  : UINT;

    bStateChanged           : BOOL;             //Indicate if state change happened
    uiInfoData_State_Prev   : UINT := 16#8;     //Previous value of Infodata.State
    bWcState_Prev           : BOOL := FALSE;    //Previous state of WcState

    //FB-s

END_VAR

(*
* ================================================================================
*                                   DESCRIPTION
* ================================================================================
* This Function Block provides connection to the Error System specifically
* for monitoring an EtherCat terminal's state of operation. The function block
* checks the content of the linked variables, that encodes the terminal's state.
* If any deviation from the nominal state is experienced an entry is created with
* all the necessary information. If the terminal goes through a series of
* different error states each state transition is tracked in a new entry.
* ================================================================================
*)

//Connect EN to EnO
EnO:=En;

IF En THEN
    //Check if pointer is OK
    IF pErrorSystem=0 THEN RETURN; END_IF

    //Any difference from normal state creates an error
    IF En AND (bWcState OR uiInfoData_State<>16#8) THEN
        bError:=TRUE;
    ELSE
        bError:=FALSE;
    END_IF

    //Change detection
    IF uiInfoData_State <> uiInfoData_State_Prev OR bWcState <> bWcState_Prev THEN
        bStateChanged := TRUE;
    ELSE
        bStateChanged := FALSE;
    END_IF

    //Update previous values
    uiInfoData_State_Prev   := uiInfoData_State;
    bWcState_Prev           := bWcState;

    //Decision tree
    IF bStateChanged THEN
        IF bError THEN
            IF ErrorData.ErrorState = DUT_ErrorState.Active THEN
                //Close active error
                //Read system time
                ErrorData.sDateTimeOff  := Tc2_EtherCat.DCTIME64_TO_STRING(Tc2_EtherCAT.F_GetActualDcTime64());
                ErrorData.ErrorState    := DUT_ErrorState.Inactive;
                //Write Off-time to Error System
                FOR nErrSysCNT := 0 TO cSizeOfErrorData - 1 DO
                    IF pErrorSystem^.aErrorData[nErrSysCNT].ErrorNum = ErrorData.ErrorNum THEN
                        pErrorSystem^.aErrorData[nErrSysCNT].sDateTimeOff   := ErrorData.sDateTimeOff;
                        pErrorSystem^.aErrorData[nErrSysCNT].ErrorState     := DUT_ErrorState.Inactive;
                        EXIT;
                    END_IF
                END_FOR

                //Clear ErrorData
                MEMSET(ADR(ErrorData), 0, SIZEOF(ErrorData));
            END_IF

            //Open a new error
            ErrorData.ErrorState    := DUT_ErrorState.Active;                                                   //Set Error State
            ErrorData.sDateTimeOn   := Tc2_EtherCat.DCTIME64_TO_STRING(Tc2_EtherCAT.F_GetActualDcTime64());     //Convert to string
            ErrorData.iTerminalID   := iTerminal_ID;                                                            //Terminal_ID

            //Error message according to uiInfoData_State and WcState
            iStateError := (uiInfoData_State AND 16#000F);                                              //Mask for operation state
            iOtherError := (uiInfoData_State AND 16#00F0);                                              //Mask for the other 3 kind of errors
            //Error messages according to the least significant digit
            CASE iStateError OF
                16#0001 :
                            ErrorData.sErrorMessage := 'Slave in INIT state;   ';
                            IF ErrorData.ErrorPriority >= 5 OR ErrorData.ErrorPriority = 0 THEN ErrorData.ErrorPriority := 5; END_IF
                16#0002 :
                            ErrorData.sErrorMessage := 'Slave in PREOP state;   ';
                            IF ErrorData.ErrorPriority >= 5 OR ErrorData.ErrorPriority = 0 THEN ErrorData.ErrorPriority := 5; END_IF
                16#0003 :
                            ErrorData.sErrorMessage := 'Slave in BOOT state;   ';
                            IF ErrorData.ErrorPriority >= 5 OR ErrorData.ErrorPriority = 0 THEN ErrorData.ErrorPriority := 5; END_IF
                16#0004 :
                            ErrorData.sErrorMessage := 'Slave in SAFEOP state;   ';
                            IF ErrorData.ErrorPriority >= 5 OR ErrorData.ErrorPriority = 0 THEN ErrorData.ErrorPriority := 5; END_IF
                16#0008 : ;                                                                             //Normal operation state
            ELSE
                ErrorData.sErrorMessage := 'Undefined State of operation;   ';
                ErrorData.sErrorMessage := CONCAT (ErrorData.sErrorMessage, UINT_TO_STRING(iStateError));
                ErrorData.sErrorMessage := CONCAT (ErrorData.sErrorMessage, '   ');
                ErrorData.ErrorPriority := 1;
            END_CASE

            //Error messages according to the second least significant digit
            CASE iOtherError OF
                16#0000 : ;                                                                         //No error case
                16#0010 :
                            ErrorData.sErrorMessage := CONCAT (ErrorData.sErrorMessage, 'Slave signals error;   ');
                            IF ErrorData.ErrorPriority >= 5 OR ErrorData.ErrorPriority = 0 THEN ErrorData.ErrorPriority := 5; END_IF
                16#0020 :
                            ErrorData.sErrorMessage := CONCAT (ErrorData.sErrorMessage, 'Invalid vendorID/productCode read;   ');
                            IF ErrorData.ErrorPriority >= 5 OR ErrorData.ErrorPriority = 0 THEN ErrorData.ErrorPriority := 5; END_IF
                16#0040 :
                            ErrorData.sErrorMessage := CONCAT (ErrorData.sErrorMessage, 'Initialisation error occured;   ');
                            IF ErrorData.ErrorPriority >= 5 OR ErrorData.ErrorPriority = 0 THEN ErrorData.ErrorPriority := 5; END_IF
            ELSE
                ErrorData.sErrorMessage := CONCAT (ErrorData.sErrorMessage, 'Undefined Error ID: ');
                ErrorData.sErrorMessage := CONCAT (ErrorData.sErrorMessage, UINT_TO_STRING(iOtherError));
                ErrorData.sErrorMessage := CONCAT (ErrorData.sErrorMessage, '   ');
                ErrorData.ErrorPriority := 1;
            END_CASE

            //Errormessage according to WcState bit
            IF bWcState THEN
                ErrorData.sErrorMessage := CONCAT (ErrorData.sErrorMessage, 'Invalid Data;');
                IF ErrorData.ErrorPriority >= 5 OR ErrorData.ErrorPriority = 0 THEN ErrorData.ErrorPriority := 5; END_IF
            END_IF

            //Check for overflow
            IF pErrorSystem^.nNoError >= cSizeOfErrorData THEN
                pErrorSystem^.nNoOverflow := pErrorSystem^.nNoOverflow+1;
            END_IF

            //Write Error Data into Error System
            ErrorData.ErrorNum  := pErrorSystem^.nNExtErrorNum ;
            MEMMOVE( ADR(pErrorSystem^.aErrorData[1]), ADR(pErrorSystem^.aErrorData[0]), (cSizeOfErrorData-1) * SIZEOF(ST_ErrorEntry));
            pErrorSystem^.aErrorData[0] := ErrorData;
            pErrorSystem^.nNExtErrorNum := pErrorSystem^.nNExtErrorNum+1;

        ELSE
            //Close Active Error
            //Read system time
            ErrorData.sDateTimeOff  := Tc2_EtherCat.DCTIME64_TO_STRING(Tc2_EtherCAT.F_GetActualDcTime64());
            ErrorData.ErrorState    := DUT_ErrorState.Inactive;
            //Write Off time to Error System
            FOR nErrSysCNT := 0 TO cSizeOfErrorData - 1 DO
                IF pErrorSystem^.aErrorData[nErrSysCNT].ErrorNum = ErrorData.ErrorNum THEN
                    pErrorSystem^.aErrorData[nErrSysCNT].sDateTimeOff   := ErrorData.sDateTimeOff;
                    pErrorSystem^.aErrorData[nErrSysCNT].ErrorState     := ErrorData.ErrorState;
                    EXIT;
                END_IF
            END_FOR

            //Clear ErrorData
            MEMSET(ADR(ErrorData), 0, SIZEOF(ErrorData));
        END_IF
    END_IF

END_IF

END_FUNCTION_BLOCK

// ---- tc_mca_std_lib/POUs/Hardware/EtherCAT_Terminals/Analog_Inputs/EL3174_0002.TcPOU
//EL3174-0002 | 4-channel analog input, -10/0...+10V, -20/0/+4...20mA, 16 bit, differential
FUNCTION_BLOCK EL3174_0002

VAR_INPUT
    En              : BOOL;
    iTerminal_ID    : INT;
    ErrorSystem     : POINTER TO ST_ErrorSystem;
END_VAR

VAR_OUTPUT
    EnO     : BOOL;
    bError  : BOOL;
END_VAR

VAR
    //Channels
    wCH1_Status     AT %I*  : WORD;
    wCH2_Status     AT %I*  : WORD;
    wCH3_Status     AT %I*  : WORD;
    wCH4_Status     AT %I*  : WORD;

    //Terminal status
    WcState_WcState AT %I*  : BOOL;
    InfoData_State  AT %I*  : UINT;

    //FB-s
    EL3174_0002_Error   : FB_TerminalError;
    CH1_Error           : FB_GenericError;
    CH2_Error           : FB_GenericError;
    CH3_Error           : FB_GenericError;
    CH4_Error           : FB_GenericError;
END_VAR

(*
* TODO: Test on hardware
*)
EnO := En;

IF En THEN
    //Channel #1 Status
    IF (wCh1_Status AND 16#2057) <> 0 THEN
        CH1_Error.sErrorMessage := 'EL3174-0002 Channel #1: ';
        IF wCH1_Status.0    THEN    CH1_Error.sErrorMessage := CONCAT(CH1_Error.sErrorMessage, 'Underrange; ');             IF CH1_Error.ErrorPriority > 100 OR CH1_Error.ErrorPriority = 0     THEN CH1_Error.ErrorPriority := 100;    END_IF      END_IF
        IF wCH1_Status.1    THEN    CH1_Error.sErrorMessage := CONCAT(CH1_Error.sErrorMessage, 'Overrange; ');              IF CH1_Error.ErrorPriority > 100 OR CH1_Error.ErrorPriority = 0     THEN CH1_Error.ErrorPriority := 100;    END_IF      END_IF
        IF wCh1_Status.2    THEN    CH1_Error.sErrorMessage := CONCAT(CH1_Error.sErrorMessage, 'Limit 1; ');                IF CH1_Error.ErrorPriority > 100 OR CH1_Error.ErrorPriority = 0     THEN CH1_Error.ErrorPriority := 100;    END_IF      END_IF
        IF wCh1_Status.4    THEN    CH1_Error.sErrorMessage := CONCAT(CH1_Error.sErrorMessage, 'Limit 2; ');                IF CH1_Error.ErrorPriority > 100 OR CH1_Error.ErrorPriority = 0     THEN CH1_Error.ErrorPriority := 100;    END_IF      END_IF
        IF wCh1_Status.6    THEN    CH1_Error.sErrorMessage := CONCAT(CH1_Error.sErrorMessage, 'Error; ');                  IF CH1_Error.ErrorPriority > 10  OR CH1_Error.ErrorPriority = 0     THEN CH1_Error.ErrorPriority := 10;     END_IF      END_IF
        IF wCh1_Status.13   THEN    CH1_Error.sErrorMessage := CONCAT(CH1_Error.sErrorMessage, 'Sync error; ');             IF CH1_Error.ErrorPriority > 10  OR CH1_Error.ErrorPriority = 0     THEN CH1_Error.ErrorPriority := 10;     END_IF      END_IF
        CH1_Error.bError := TRUE;
    ELSE
        CH1_Error.bError        := FALSE;
        CH1_Error.sErrorMessage := '';
    END_IF

    //Channel #2 Status
    IF (wCh2_Status AND 16#2057) <> 0 THEN
        CH2_Error.sErrorMessage := 'EL3174-0002 Channel #2: ';
        IF wCH2_Status.0    THEN    CH2_Error.sErrorMessage := CONCAT(CH2_Error.sErrorMessage, 'Underrange; ');             IF CH2_Error.ErrorPriority > 100 OR CH2_Error.ErrorPriority = 0     THEN CH2_Error.ErrorPriority := 100;    END_IF      END_IF
        IF wCH2_Status.1    THEN    CH2_Error.sErrorMessage := CONCAT(CH2_Error.sErrorMessage, 'Overrange; ');              IF CH2_Error.ErrorPriority > 100 OR CH2_Error.ErrorPriority = 0     THEN CH2_Error.ErrorPriority := 100;    END_IF      END_IF
        IF wCh2_Status.2    THEN    CH2_Error.sErrorMessage := CONCAT(CH2_Error.sErrorMessage, 'Limit 1; ');                IF CH2_Error.ErrorPriority > 100 OR CH2_Error.ErrorPriority = 0     THEN CH2_Error.ErrorPriority := 100;    END_IF      END_IF
        IF wCh2_Status.4    THEN    CH2_Error.sErrorMessage := CONCAT(CH2_Error.sErrorMessage, 'Limit 2; ');                IF CH2_Error.ErrorPriority > 100 OR CH2_Error.ErrorPriority = 0     THEN CH2_Error.ErrorPriority := 100;    END_IF      END_IF
        IF wCh2_Status.6    THEN    CH2_Error.sErrorMessage := CONCAT(CH2_Error.sErrorMessage, 'Error; ');                  IF CH2_Error.ErrorPriority > 10  OR CH2_Error.ErrorPriority = 0     THEN CH2_Error.ErrorPriority := 10;     END_IF      END_IF
        IF wCh2_Status.13   THEN    CH2_Error.sErrorMessage := CONCAT(CH2_Error.sErrorMessage, 'Sync error; ');             IF CH2_Error.ErrorPriority > 10  OR CH2_Error.ErrorPriority = 0     THEN CH2_Error.ErrorPriority := 10;     END_IF      END_IF
        CH2_Error.bError := TRUE;
    ELSE
        CH2_Error.bError        := FALSE;
        CH2_Error.sErrorMessage := '';
    END_IF

    //Channel #3 Status
    IF (wCh3_Status AND 16#2057) <> 0 THEN
        CH3_Error.sErrorMessage := 'EL3174-0002 Channel #3: ';
        IF wCH3_Status.0    THEN    CH3_Error.sErrorMessage := CONCAT(CH3_Error.sErrorMessage, 'Underrange; ');             IF CH3_Error.ErrorPriority > 100 OR CH3_Error.ErrorPriority = 0     THEN CH3_Error.ErrorPriority := 100;    END_IF      END_IF
        IF wCH3_Status.1    THEN    CH3_Error.sErrorMessage := CONCAT(CH3_Error.sErrorMessage, 'Overrange; ');              IF CH3_Error.ErrorPriority > 100 OR CH3_Error.ErrorPriority = 0     THEN CH3_Error.ErrorPriority := 100;    END_IF      END_IF
        IF wCh3_Status.2    THEN    CH3_Error.sErrorMessage := CONCAT(CH3_Error.sErrorMessage, 'Limit 1; ');                IF CH3_Error.ErrorPriority > 100 OR CH3_Error.ErrorPriority = 0     THEN CH3_Error.ErrorPriority := 100;    END_IF      END_IF
        IF wCh3_Status.4    THEN    CH3_Error.sErrorMessage := CONCAT(CH3_Error.sErrorMessage, 'Limit 2; ');                IF CH3_Error.ErrorPriority > 100 OR CH3_Error.ErrorPriority = 0     THEN CH3_Error.ErrorPriority := 100;    END_IF      END_IF
        IF wCh3_Status.6    THEN    CH3_Error.sErrorMessage := CONCAT(CH3_Error.sErrorMessage, 'Error; ');                  IF CH3_Error.ErrorPriority > 10  OR CH3_Error.ErrorPriority = 0     THEN CH3_Error.ErrorPriority := 10;     END_IF      END_IF
        IF wCh3_Status.13   THEN    CH3_Error.sErrorMessage := CONCAT(CH3_Error.sErrorMessage, 'Sync error; ');             IF CH3_Error.ErrorPriority > 10  OR CH3_Error.ErrorPriority = 0     THEN CH3_Error.ErrorPriority := 10;     END_IF      END_IF
        CH3_Error.bError := TRUE;
    ELSE
        CH3_Error.bError        := FALSE;
        CH3_Error.sErrorMessage := '';
    END_IF

    //Channel #4 Status
    IF (wCh4_Status AND 16#2057) <> 0 THEN
        CH4_Error.sErrorMessage := 'EL3174-0002 Channel #4: ';
        IF wCH4_Status.0    THEN    CH4_Error.sErrorMessage := CONCAT(CH4_Error.sErrorMessage, 'Underrange; ');             IF CH4_Error.ErrorPriority > 100 OR CH4_Error.ErrorPriority = 0     THEN CH4_Error.ErrorPriority := 100;    END_IF      END_IF
        IF wCH4_Status.1    THEN    CH4_Error.sErrorMessage := CONCAT(CH4_Error.sErrorMessage, 'Overrange; ');              IF CH4_Error.ErrorPriority > 100 OR CH4_Error.ErrorPriority = 0     THEN CH4_Error.ErrorPriority := 100;    END_IF      END_IF
        IF wCh4_Status.2    THEN    CH4_Error.sErrorMessage := CONCAT(CH4_Error.sErrorMessage, 'Limit 1; ');                IF CH4_Error.ErrorPriority > 100 OR CH4_Error.ErrorPriority = 0     THEN CH4_Error.ErrorPriority := 100;    END_IF      END_IF
        IF wCh4_Status.4    THEN    CH4_Error.sErrorMessage := CONCAT(CH4_Error.sErrorMessage, 'Limit 2; ');                IF CH4_Error.ErrorPriority > 100 OR CH4_Error.ErrorPriority = 0     THEN CH4_Error.ErrorPriority := 100;    END_IF      END_IF
        IF wCh4_Status.6    THEN    CH4_Error.sErrorMessage := CONCAT(CH4_Error.sErrorMessage, 'Error; ');                  IF CH4_Error.ErrorPriority > 10  OR CH4_Error.ErrorPriority = 0     THEN CH4_Error.ErrorPriority := 10;     END_IF      END_IF
        IF wCh4_Status.13   THEN    CH4_Error.sErrorMessage := CONCAT(CH4_Error.sErrorMessage, 'Sync error; ');             IF CH4_Error.ErrorPriority > 10  OR CH4_Error.ErrorPriority = 0     THEN CH4_Error.ErrorPriority := 10;     END_IF      END_IF
        CH4_Error.bError := TRUE;
    ELSE
        CH4_Error.bError        := FALSE;
        CH4_Error.sErrorMessage := '';
    END_IF

END_IF



//Error FB instance
EL3174_0002_Error(
    En                  := TRUE,
    iTerminal_ID        := iTerminal_ID,
    bWcState            := WcState_WcState,
    uiInfoData_State    := InfoData_State,
    pErrorSystem        := ErrorSystem,
    bError              => bError,
);

CH1_Error (
    En              := En,
    bError          := ,
    sErrorMessage   := ,
    ErrorPriority   := ,
    iTerminal_ID    := iTerminal_ID,
    pErrorSystem    := ErrorSystem,
    EnO             => ,
);

CH2_Error (
    En              := En,
    bError          := ,
    sErrorMessage   := ,
    ErrorPriority   := ,
    iTerminal_ID    := iTerminal_ID,
    pErrorSystem    := ErrorSystem,
    EnO             => ,
);

CH3_Error (
    En              := En,
    bError          := ,
    sErrorMessage   := ,
    ErrorPriority   := ,
    iTerminal_ID    := iTerminal_ID,
    pErrorSystem    := ErrorSystem,
    EnO             => ,
);

CH4_Error (
    En              := En,
    bError          := ,
    sErrorMessage   := ,
    ErrorPriority   := ,
    iTerminal_ID    := iTerminal_ID,
    pErrorSystem    := ErrorSystem,
    EnO             => ,
);

END_FUNCTION_BLOCK

// ---- tc_mca_std_lib/POUs/Hardware/EtherCAT_Terminals/Analog_Inputs/EL3214.TcPOU
//EL3214 | 4-channel analog input terminal, PT100 (RTD)
FUNCTION_BLOCK EL3214

VAR_INPUT
    En              : BOOL;
    iTerminal_ID    : INT;
    ErrorSystem     : POINTER TO ST_ErrorSystem;
END_VAR

VAR_OUTPUT
    EnO     : BOOL;
    bError  : BOOL;
END_VAR

VAR
    //Channels
    wCh1_Status     AT %I* : WORD;
    wCh2_Status     AT %I* : WORD;
    wCh3_Status     AT %I* : WORD;
    wCh4_Status     AT %I* : WORD;

    //Terminal status
    WcState_WcState     AT %I*: BOOL;
    InfoData_State      AT %I*: UINT;

    //FB-s
    EL3214_Error    : FB_TerminalError;
    CH1_Error       : FB_GenericError;
    CH2_Error       : FB_GenericError;
    CH3_Error       : FB_GenericError;
    CH4_Error       : FB_GenericError;
END_VAR

(*
* TODO: Test on hardware
*)

EnO := En;

//Channel #1 Status
IF (wCh1_Status AND 16#0043) <> 0 THEN
    CH1_Error.sErrorMessage := 'EL3214 Channel #1: ';
    IF wCh1_Status.0    THEN    CH1_Error.sErrorMessage := CONCAT(CH1_Error.sErrorMessage, 'Underrange; ');             IF CH1_Error.ErrorPriority > 100 OR CH1_Error.ErrorPriority = 0     THEN CH1_Error.ErrorPriority := 100;    END_IF      END_IF
    IF wCh1_Status.1    THEN    CH1_Error.sErrorMessage := CONCAT(CH1_Error.sErrorMessage, 'Overrange; ');              IF CH1_Error.ErrorPriority > 100 OR CH1_Error.ErrorPriority = 0     THEN CH1_Error.ErrorPriority := 100;    END_IF      END_IF
    IF wCh1_Status.6    THEN    CH1_Error.sErrorMessage := CONCAT(CH1_Error.sErrorMessage, 'Error; ');                  IF CH1_Error.ErrorPriority > 10  OR CH1_Error.ErrorPriority = 0     THEN CH1_Error.ErrorPriority := 10;     END_IF      END_IF
    CH1_Error.bError := TRUE;
ELSE
    CH1_Error.bError := FALSE;
    CH1_Error.sErrorMessage := '';
END_IF

//Channel #2 Status
IF (wCh2_Status AND 16#0043) <> 0 THEN
    CH2_Error.sErrorMessage := 'EL3214 Channel #2: ';
    IF wCh2_Status.0    THEN    CH2_Error.sErrorMessage := CONCAT(CH2_Error.sErrorMessage, 'Underrange; ');             IF CH2_Error.ErrorPriority > 100 OR CH2_Error.ErrorPriority = 0     THEN CH2_Error.ErrorPriority := 100;    END_IF      END_IF
    IF wCh2_Status.1    THEN    CH2_Error.sErrorMessage := CONCAT(CH2_Error.sErrorMessage, 'Overrange; ');              IF CH2_Error.ErrorPriority > 100 OR CH2_Error.ErrorPriority = 0     THEN CH2_Error.ErrorPriority := 100;    END_IF      END_IF
    IF wCh2_Status.6    THEN    CH2_Error.sErrorMessage := CONCAT(CH2_Error.sErrorMessage, 'Error; ');                  IF CH2_Error.ErrorPriority > 10  OR CH2_Error.ErrorPriority = 0     THEN CH2_Error.ErrorPriority := 10;     END_IF      END_IF
    CH2_Error.bError := TRUE;
ELSE
    CH2_Error.bError := FALSE;
    CH2_Error.sErrorMessage := '';
END_IF

//Channel #3 Status
IF (wCh3_Status AND 16#0043) <> 0 THEN
    CH3_Error.sErrorMessage := 'EL3214 Channel #3: ';
    IF wCh3_Status.0    THEN    CH3_Error.sErrorMessage := CONCAT(CH3_Error.sErrorMessage, 'Underrange; ');             IF CH3_Error.ErrorPriority > 100 OR CH3_Error.ErrorPriority = 0     THEN CH3_Error.ErrorPriority := 100;    END_IF      END_IF
    IF wCh3_Status.1    THEN    CH3_Error.sErrorMessage := CONCAT(CH3_Error.sErrorMessage, 'Overrange; ');              IF CH3_Error.ErrorPriority > 100 OR CH3_Error.ErrorPriority = 0     THEN CH3_Error.ErrorPriority := 100;    END_IF      END_IF
    IF wCh3_Status.6    THEN    CH3_Error.sErrorMessage := CONCAT(CH3_Error.sErrorMessage, 'Error; ');                  IF CH3_Error.ErrorPriority > 10  OR CH3_Error.ErrorPriority = 0     THEN CH3_Error.ErrorPriority := 10;     END_IF      END_IF
    CH3_Error.bError := TRUE;
ELSE
    CH3_Error.bError := FALSE;
    CH3_Error.sErrorMessage := '';
END_IF

//Channel #4 Status
IF (wCh4_Status AND 16#0043) <> 0 THEN
    CH4_Error.sErrorMessage := 'EL3214 Channel #4: ';
    IF wCh4_Status.0    THEN    CH4_Error.sErrorMessage := CONCAT(CH4_Error.sErrorMessage, 'Underrange; ');             IF CH4_Error.ErrorPriority > 100 OR CH4_Error.ErrorPriority = 0     THEN CH4_Error.ErrorPriority := 100;    END_IF      END_IF
    IF wCh4_Status.1    THEN    CH4_Error.sErrorMessage := CONCAT(CH4_Error.sErrorMessage, 'Overrange; ');              IF CH4_Error.ErrorPriority > 100 OR CH4_Error.ErrorPriority = 0     THEN CH4_Error.ErrorPriority := 100;    END_IF      END_IF
    IF wCh4_Status.6    THEN    CH4_Error.sErrorMessage := CONCAT(CH4_Error.sErrorMessage, 'Error; ');                  IF CH4_Error.ErrorPriority > 10  OR CH4_Error.ErrorPriority = 0     THEN CH4_Error.ErrorPriority := 10;     END_IF      END_IF
    CH4_Error.bError := TRUE;
ELSE
    CH4_Error.bError := FALSE;
    CH4_Error.sErrorMessage := '';
END_IF

//Error FB instance
EL3214_Error(
    En                  := TRUE,
    iTerminal_ID        := iTerminal_ID,
    bWcState            := WcState_WcState,
    uiInfoData_State    := InfoData_State,
    pErrorSystem        := ErrorSystem,
    bError              => bError,
);

CH1_Error (
    En              := En,
    bError          := ,
    sErrorMessage   := ,
    ErrorPriority   := ,
    iTerminal_ID    := iTerminal_ID,
    pErrorSystem    := ErrorSystem,
    EnO             => ,
);

CH2_Error (
    En              := En,
    bError          := ,
    sErrorMessage   := ,
    ErrorPriority   := ,
    iTerminal_ID    := iTerminal_ID,
    pErrorSystem    := ErrorSystem,
    EnO             => ,
);

CH3_Error (
    En              := En,
    bError          := ,
    sErrorMessage   := ,
    ErrorPriority   := ,
    iTerminal_ID    := iTerminal_ID,
    pErrorSystem    := ErrorSystem,
    EnO             => ,
);

CH4_Error (
    En              := En,
    bError          := ,
    sErrorMessage   := ,
    ErrorPriority   := ,
    iTerminal_ID    := iTerminal_ID,
    pErrorSystem    := ErrorSystem,
    EnO             => ,
);

END_FUNCTION_BLOCK

// ---- tc_mca_std_lib/POUs/Hardware/EtherCAT_Terminals/Analog_Inputs/EL3255.TcPOU
//EL3255 | 5-channel potentiometer measurement with sensor supply
FUNCTION_BLOCK EL3255

VAR_INPUT
    En              : BOOL;
    iTerminal_ID    : INT;
    ErrorSystem     : POINTER TO ST_ErrorSystem;
END_VAR

VAR_OUTPUT
    EnO     : BOOL;
    bError  : BOOL;
END_VAR

VAR
    wCH1_Status     AT %I*  : WORD;
    wCH2_Status     AT %I*  : WORD;
    wCH3_Status     AT %I*  : WORD;
    wCH4_Status     AT %I*  : WORD;
    wCH5_Status     AT %I*  : WORD;
    WcState_WcState AT %I*  : BOOL;
    InfoData_State  AT %I*  : UINT;

